// TwinCAT 3 PLC project Untitled1
// ProgramVersion: 3.1.4023.0
// CompilerDefines: VISU_USEWSTRING
// libraries:
//   CmpBitmapPool, * (System)
//   Tc2_Standard, * (Beckhoff Automation GmbH)
//   Tc2_System, * (Beckhoff Automation GmbH)
//   Tc3_Module, * (Beckhoff Automation GmbH)
//   VisuDialogs, * (System)
//   MachineManage,newest,Secote
// project tree:
//   DUTs/ E_Axis.TcDUT, E_Cylinder.TcDUT, E_Line.TcDUT, E_LineClose.TcDUT, E_LoadClose.TcDUT, E_LoadPriority.TcDUT, E_MachineType.TcDUT, E_Station.TcDUT, E_TakeMode.TcDUT, ST_Input.TcDUT, ST_Output.TcDUT, ST_Recipe.TcDUT, ST_Setting.TcDUT
//   DUTs/Station/Dismantling/ ST_StationDismantling.TcDUT, ST_StationDismantlingHandshake.TcDUT
//   DUTs/Station/ E_StationState.TcDUT, ST_StationHandshake.TcDUT, ST_StationParameter.TcDUT
//   DUTs/Station/Line0Buffer/ ST_StationLine0Buffer.TcDUT, ST_StationLine0BufferHandshake.TcDUT
//   DUTs/Station/Line0Load/ ST_StationLine0Load.TcDUT, ST_StationLine0LoadHandshake.TcDUT
//   DUTs/Station/LineLoad/ ST_StationLineLoad.TcDUT, ST_StationLineLoadHandshake.TcDUT
//   DUTs/Station/TakeLoad/ ST_StationTakeLoad.TcDUT, ST_StationTakeLoadHandshake.TcDUT
//   DUTs/Station/UnloadElevator/ ST_StationUnloadElevator.TcDUT, ST_StationUnloadElevatorHandshake.TcDUT
//   DUTs/Station/UnloadLine/ ST_StationUnloadLine.TcDUT, ST_StationUnloadLineHandshake.TcDUT
//   DUTs/Station/UnloadUc/ ST_StationUnloadUc.TcDUT, ST_StationUnloadUcHandshake.TcDUT
//   DUTs/Station/UnloadUc_311/ ST_StationUnloadUc_311.TcDUT, ST_StationUnloadUc_311Handshake.TcDUT
//   / GlobalTextList.TcGTLO, PlcTask.TcTTO, RecipeManager.TcRMO (not stored), VISU_TASK.TcTTO, 视图管理器.TcVMO (not stored)
//   GVLs/ GVL.TcGVL, GVL_Data.TcGVL, GVL_IO.TcGVL
//   POUs/Device/ FB_LineAxis.TcPOU
//   POUs/ MAIN.TcPOU, P_Alarm.TcPOU, P_Device.TcPOU, P_Station.TcPOU, P_System.TcPOU
//   POUs/Station/ FB_StationDismantling.TcPOU, FB_StationLine0Buffer.TcPOU, FB_StationLine0Load.TcPOU, FB_StationLineLoad.TcPOU, FB_StationTakeLoad.TcPOU, FB_StationUnloadElevator.TcPOU, FB_StationUnloadLine.TcPOU, FB_StationUnloadUc.TcPOU, FB_StationUnLoadUc_311.TcPOU
//   VISUs/Ctrl/ CtrlLine.TcVIS, CtrlOther.TcVIS, CtrlOutput.TcVIS, CtrlInput.TcVIS, FrameMain.TcVIS
//   VISUs/Image/ ImagePool.TcIPO (not stored)
//   VISUs/ PageData.TcVIS, PageHome.TcVIS, PageMessage.TcVIS, PageMonitor.TcVIS, PageSetting.TcVIS
//   VISUs/Text/ InputText.TcTLO, LineClose.TcTLO, LineLoadClose.TcTLO, LoadPriority.TcTLO, MachineType.TcTLO, ManualText.TcTLO, OutputText.TcTLO

CONFIGURATION Untitled1
    RESOURCE PLC ON TwinCAT3
        TASK PlcTask(INTERVAL := T#2ms, PRIORITY := 20);
        TASK VISU_TASK(INTERVAL := T#50000us, PRIORITY := 30);
        PROGRAM MAIN WITH PlcTask : MAIN;
        PROGRAM VisuElems_Visu_Prg WITH VISU_TASK : VisuElems.Visu_Prg;
    END_RESOURCE
END_CONFIGURATION

// ---- DUTs/E_Axis.TcDUT
{attribute 'qualified_only'}
{attribute 'strict'}
TYPE E_Axis :
(
	TakeY:=1,
	TakeZ,
	UC_Y
);
END_TYPE

// ---- DUTs/E_Cylinder.TcDUT
{attribute 'qualified_only'}
{attribute 'strict'}
TYPE E_Cylinder :
(
Line0Part:=1,//主流线分料气缸

Line0Prevent,//主流线阻挡气缸

Line1Elevator,//流水线1提升气缸

Line1Lift,//流水线1顶升气缸

Line1Prevent,//流水线1阻挡气缸

Line1Rotate,//流水线1旋转气缸

Line1Adjust1,//流水线1调宽气缸1

Line2Lift,//流水线2顶升气缸

Line2Prevent,//流水线2阻挡气缸

Line2Standard1,//流水线2校平气缸1

Line2Standard2,//流水线2校平气缸2

Line2OpenLateral1,//流水线2解锁侧推气缸1

Line2OpenRotate,//流水线2解锁旋转气缸

Line2OpenLateral2,//流水线2解锁侧推气缸2

Line3LoadLift,//流水线3上料位顶升

Line3LoadPrevent,//流水线3上料位阻挡

Line3LoadRotate,//流水线3上料位旋转

Line3OpenLift,//流水线3解锁位顶升

Line3OpenPrevent,//流水线3解锁位阻挡

Line3Standard1,//流水线3校平气缸1

Line3Standard2,//流水线3校平气缸2

Line3OpenLateral1,//流水线3解锁侧推气缸1

Line3OpenRotate,//流水线3解锁旋转气缸

Line3OpenLateral2,//流水线3解锁侧推气缸2

TakeLift1,//取料模组升降气缸1

TakeLift2,//取料模组升降气缸2

TakeClamp,//取料模组夹紧气缸

UcLift,//下UC模组升降气缸

UcClamp,//下UC模组夹紧气缸

UcSwing,//下UC模组摆动气缸

UcLift1,//下UC升降气缸1

UcClamp1,//下UC夹紧气缸1

UcRotate1,//下UC旋转气缸1

UcLift2,//下UC升降气缸2

UcClamp2,//下UC夹紧气缸2

UcRotate2,//下UC旋转气缸2

UcDrive,//下UC皮带推料气缸

FrockElevator1,//下工装提升气缸1

FrockRotateDown1,//下工装旋转压紧气缸1

FrockPush1,//下工装拨料气缸1

FrockElevator2,//下工装提升气缸2

FrockRotateDown2,//下工装旋转压紧气缸2

FrockPush2,//下工装拨料气缸2

FrockBelt//下工装皮带推料气缸
);
END_TYPE

// ---- DUTs/E_Line.TcDUT
{attribute 'qualified_only'}
{attribute 'strict'}
TYPE E_Line :
(
	UnloadElevator := 1,
	UnloadUC,
	Line1,
	Line2,
	Line3
	
);
END_TYPE

// ---- DUTs/E_LineClose.TcDUT
{attribute 'qualified_only'}
{attribute 'strict'}
TYPE E_LineClose :
(
	None := 0,
	Line2,
	Line3
);
END_TYPE

// ---- DUTs/E_LoadClose.TcDUT
{attribute 'qualified_only'}
{attribute 'strict'}
TYPE E_LoadClose :
(
	None:=0,// 不关闭
	Line0,
	Line1
);
END_TYPE

// ---- DUTs/E_LoadPriority.TcDUT
{attribute 'qualified_only'}
{attribute 'strict'}
TYPE E_LoadPriority :
(
	None := 0,// 无等级
	Line0,// 优先0
	Line1// 优先1
);
END_TYPE

// ---- DUTs/E_MachineType.TcDUT
{attribute 'qualified_only'}
{attribute 'strict'}
TYPE E_MachineType :
(
	None:=0,
	RH353,
	RH367,
	RH311,
	RH201,
	RH069,
	RH373,
	LH353,
	LH367,
	LH311,
	LH201,
	LH069,
	LH373
);
END_TYPE

// ---- DUTs/E_Station.TcDUT
{attribute 'qualified_only'}
{attribute 'strict'}
TYPE E_Station :
(
	Line0Load:=0,// 主流线上料工站
	Line0Buffer,// 主流线缓存工站
	TakeLoad,// 上料取料工站
	Line3Load,// 流线3上料工站
	Line1Load,// 流线2上料工站
	Line2Dismantling,// 流线2拆解工站
	Line3Dismantling,// 流线3拆解工站
	Line2UnloadElevator,// 线体2下工装
	Line3UnloadElevator,// 线体3下工装
	Line2UnloadUc,// 线体2 下UC
	Line3UnloadUc,// 线体2 下UC
	UnloadLineUc,// 下UC 线体
	UnloadLineElevator,// 下工装 线体
	UnloadUc_311,// 下UC模组
	Length
);
END_TYPE

// ---- DUTs/E_TakeMode.TcDUT
{attribute 'qualified_only'}
{attribute 'strict'}
TYPE E_TakeMode :
(
	None := 0,// 不动作
	Take0,// 取Line0料
	Take1,// 取Line1料
	Take3Load,// 取Line3上料站 产品
	Place1,// 放Line1料
	Place3Load// 放线体3上料站
);
END_TYPE

// ---- DUTs/Station/Dismantling/ST_StationDismantling.TcDUT
TYPE ST_StationDismantling :
STRUCT
	fbLift:				 	REFERENCE TO FB_Cylinder;// 顶升气缸
	fbPrevent:				REFERENCE TO FB_Cylinder;// 阻挡气缸
	fbStandard1:			REFERENCE TO FB_Cylinder;// 校平气缸1
	fbStandard2:			REFERENCE TO FB_Cylinder;// 校平气缸2
	fbLateral1:				REFERENCE TO FB_Cylinder;// 侧推气缸1
	fbLateral2:				REFERENCE TO FB_Cylinder;// 侧推气缸2
	fbRotate:				REFERENCE TO FB_Cylinder;// 旋转气缸
	bPalletCheck1:			BOOL;// 流入光电
	bPalletCheck2:			BOOL;// 到位光电
	bPalletCheck3:			BOOL;// 流出光电
	eState:					E_StationState;
	bClose:					BOOL;// 关闭线体
	bCloseUnloadElevator:	BOOL;// 关闭下工装
	stHandshake:			ST_StationDismantlingHandshake;
END_STRUCT
END_TYPE

// ---- DUTs/Station/Dismantling/ST_StationDismantlingHandshake.TcDUT
TYPE ST_StationDismantlingHandshake :
STRUCT
	bRequestLineLoad_D:			BOOL;// 拆解工站 请求上料 只写
	bResponseDismantling_D:		BOOL;// 收到 拆解工站 请求上料 只读
	
	bRequestUc:					BOOL;// 拆解站 向下UC站 请求放料 只写
	bResponseDismantling_Uc:	BOOL;// 收到 拆解站 向下UC站 请求放料 只读
	
	bRequestElevator:			BOOL;// 拆解站 向下工装 请求放料 只写
	bResponseDismantling_E:		BOOL;// 收到 拆解站 向下工装站 请求放料 只读
	
END_STRUCT
END_TYPE

// ---- DUTs/Station/E_StationState.TcDUT
{attribute 'qualified_only'}
{attribute 'strict'}
TYPE E_StationState :
(
	None:=0,
	Load,// 等待上料
	Busy,// 工作中
	Done// 工作完成
);
END_TYPE

// ---- DUTs/Station/Line0Buffer/ST_StationLine0Buffer.TcDUT
TYPE ST_StationLine0Buffer :
STRUCT
	bPlace:				BOOL;// 到位光电
	eState:				E_StationState;
	stHandshake:		ST_StationLine0BufferHandshake;
END_STRUCT
END_TYPE

// ---- DUTs/Station/Line0Buffer/ST_StationLine0BufferHandshake.TcDUT
TYPE ST_StationLine0BufferHandshake :
STRUCT
	bRequestLine0Load:			BOOL;// 请求线体0 上料站 放料 只写
	bResponseLine0Buffer:		BOOL;// 收到线体0 上料缓存站 放料请求 只读
	
	bRequestLine0Buffer_T:		BOOL;// 取料站 向线体0 请求 取料 只读
	bResponseTake_T:			BOOL;// 收到 取料站 取料请求 只写
END_STRUCT
END_TYPE

// ---- DUTs/Station/Line0Load/ST_StationLine0Load.TcDUT
TYPE ST_StationLine0Load :
STRUCT
	fbPart:			REFERENCE TO FB_Cylinder;// 分料气缸
	fbPrevent:		REFERENCE TO FB_Cylinder;// 阻挡气缸
	bPartCheck:		BOOL;// 分料光电
	bPreventCheck:	BOOL;// 阻挡光电
	stHandshake:	ST_StationLine0LoadHandshake;	
END_STRUCT
END_TYPE

// ---- DUTs/Station/Line0Load/ST_StationLine0LoadHandshake.TcDUT
TYPE ST_StationLine0LoadHandshake :
STRUCT
	bRequestLine0Load:			BOOL;// 请求线体0 上料站 放料 只读
	bResponseLine0Buffer:		BOOL;// 收到线体0 上料缓存站 放料请求 只写
END_STRUCT
END_TYPE

// ---- DUTs/Station/LineLoad/ST_StationLineLoad.TcDUT
TYPE ST_StationLineLoad :
STRUCT
	fbElevator:				REFERENCE TO FB_Cylinder;// 提升气缸
	fbLift:					REFERENCE TO FB_Cylinder;// 顶升气缸
	fbPrevent:				REFERENCE TO FB_Cylinder;// 阻挡气缸
	fbRotate:				REFERENCE TO FB_Cylinder;// 旋转气缸
	fbAdjust1:				REFERENCE TO FB_Cylinder;// 调宽气缸
	bPalletCheck1:			BOOL;// 流入光电
	bPalletCheck2:			BOOL;// 到位光电
	bPalletCheck3:			BOOL;// 流出光电
	eState:					E_StationState;
	bIsClosed:				BOOL;// 线体关闭
	bIsTaking:				BOOL;// 取料站 取料中
	bIsPlacing:				BOOL;// 取料站 放料中
	bManualLoad:			BOOL;// 手动上料 
	stHandshake:			ST_StationLineLoadHandshake;
END_STRUCT
END_TYPE

// ---- DUTs/Station/LineLoad/ST_StationLineLoadHandshake.TcDUT
TYPE ST_StationLineLoadHandshake :
STRUCT
	bRequestLineLoad_T:			BOOL;// 取料站 请求取料 只读
	bResponseTake_T:			BOOL;// 收到 取料站 请求取料 只写
	
	bRequestLineLoad_P:			BOOL;// 取料站 请求放料 只读
	bResponseTake_P:			BOOL;// 收到 取料站 请求放料 只写
	
	bRequestTake_P_M:			BOOL;// 上游设备 请求放料 只读
	bResponseMachine_P:			BOOL;// 收到 上游设备 请求放料 只写
	
	bRequestLineLoad_D:			BOOL;// 拆解工站 请求上料 只读
	bResponseDismantling_D:		BOOL;// 收到 拆解工站 请求上料 只写
END_STRUCT
END_TYPE

// ---- DUTs/Station/ST_StationHandshake.TcDUT
TYPE ST_StationHandshake :
STRUCT
	(*bLine0BufferRequestLine0Load:			BOOL;// Line0缓存站 请求上料站放料
	bLine0LoadResponseLine0Buffer:			BOOL;// line0上料站 收到缓存站请求
	

	arrRequestTaskLine:						ARRAY[0..2] OF	BOOL;// 请求取线体上料站 产品 0:Lin0 1:Line1 2:Lin3Load
	arrRequestPlaceLine:					ARRAY[1..2] OF	BOOL;// 请求往线体上料站 放料 1:Line1 2:Lin3Load
	
	arrResponseTaskLine:					ARRAY[0..2] OF	BOOL;// 线体上料站收到取料请求 0:Lin0 1:Line1 2:Lin3Load
	arrResponsePlaceLine:					ARRAY[1..2] OF 	BOOL;// 线体上料站收到放料请求 1:Line1 2:Lin3Load
	
	
	bLoadMachineReady:					    BOOL;// Line1对接设备准备就绪
	bLoadMachineReadyOk:					BOOL;// 收到Line1对接设备请求信号
	
	arrDismantlingRequest:					ARRAY[1..2] OF BOOL;// 拆解站请求放料 1:Line2 2:Lin3
	arrDismantlingResponse:					ARRAY[1..2] OF BOOL;// 上料站收到拆解站请求信号 1:Line1 2:Lin3
	
	arrDismantlingRequestUc:				ARRAY[1..2] OF BOOL;// 拆解站请求取Uc 1:Line2 2:Lin3
	arrDismantlingResponseUc:				ARRAY[1..2] OF BOOL;// 收到拆解站请求取Uc 1:Line2 2:Lin3
	
	arrUnloadUcRequest:						ARRAY[1..2] OF BOOL;// 下UC工站 请求放料
	arrUnloadUcResponse:					ARRAY[1..2] OF BOOL;// 下UC线体 收到放料请求
	
	arrUnloadElevatorRequest:				ARRAY[1..2] OF BOOL;// 下UC工站 请求放料
	arrUnloadElevatorResponse:				ARRAY[1..2] OF BOOL;// 下UC线体 收到放料请求*)
END_STRUCT
END_TYPE

// ---- DUTs/Station/ST_StationParameter.TcDUT
TYPE ST_StationParameter :
STRUCT
	stLine0Load:			ST_StationLine0Load;// 主流线上料工站
	stLine0Buffer:			ST_StationLine0Buffer;// 主流线缓存工站
	stTakeLoad:				ST_StationTakeLoad;// 上料取料工站
	stLine3Load:			ST_StationLineLoad;// 流线3上料工站
	stLine1Load:			ST_StationLineLoad;// 流线2上料工站
	stLine2Dismantling:		ST_StationDismantling;// 流线2拆解工站
	stLine3Dismantling:		ST_StationDismantling;// 流线3拆解工站
	stLine2UnloadElevator:	ST_StationUnloadElevator;// 线体2下工装
	stLine3UnloadElevator:	ST_StationUnloadElevator;// 线体3下工装
	stLine2UnloadUc:		ST_StationUnloadUc;// 线体2 下UC
	stLine3UnloadUc:		ST_StationUnloadUc;// 线体2 下UC
	stUnloadLineUc:			ST_StationUnloadLine;// 下UC 线体
	stUnloadLineElevator:	ST_StationUnloadLine;// 下工装 线体
	stUnloadUc_311:			ST_StationUnloadUc_311;// 下UC 模组
END_STRUCT
END_TYPE

// ---- DUTs/Station/TakeLoad/ST_StationTakeLoad.TcDUT
TYPE ST_StationTakeLoad :
STRUCT
	fbTakeLift1:		REFERENCE TO FB_Cylinder;// 升降气缸1
	fbTakeLift2:		REFERENCE TO FB_Cylinder;// 升降气缸2
	fbTakeClamp:		REFERENCE TO FB_Cylinder;// 加紧气缸
	fbTakeZ:			REFERENCE TO FB_Axis;// Z轴
	fbTakeY:			REFERENCE TO FB_Axis;// Y轴
	eState:				E_StationState;
	stHandshake:		ST_StationTakeLoadHandshake;
END_STRUCT
END_TYPE

// ---- DUTs/Station/TakeLoad/ST_StationTakeLoadHandshake.TcDUT
TYPE ST_StationTakeLoadHandshake :
STRUCT
	bRequestLine0Buffer_T0:		BOOL;// 取料站 向线体0 请求 取料 只写
	bResponseTake_T0:			BOOL;// 收到 取料站 取料请求 只读
	
	bRequestLineLoad_T1:	BOOL;// 取料站 请求取料 Line1 只写
	bResponseTake_T1:		BOOL;// 收到 取料站 请求取料 Line1 只读
	
	bRequestLineLoad_T3:	BOOL;// 取料站 请求取料 Line2 只写
	bResponseTake_T3:		BOOL;// 收到 取料站 请求取料 Line3 只读
	
	bRequestLineLoad_P3:	BOOL;// 取料站 请求放料 Lin3 只写
	bResponseTake_P3:		BOOL;// 收到 取料站 请求放料 Line3 只读
	
	bRequestLineLoad_P1:	BOOL;// 取料站 请求放料 Lin1 只写
	bResponseTake_P1:		BOOL;// 收到 取料站 请求放料 Line1 只读
END_STRUCT
END_TYPE

// ---- DUTs/Station/UnloadElevator/ST_StationUnloadElevator.TcDUT
TYPE ST_StationUnloadElevator :
STRUCT
	bFrockElevator1NoneCheck:			BOOL;//工装有无检测
	fbFrockElevator:					REFERENCE TO FB_Cylinder;// 提升气缸
	fbFrockRotateDown:					REFERENCE TO FB_Cylinder;// 旋转压紧气缸
	fbFrockPush:						REFERENCE TO FB_Cylinder;// 拨料气缸
	bManualUnload:						BOOL;// 手动下料
	stHandshake:						ST_StationUnloadElevatorHandshake;
END_STRUCT
END_TYPE

// ---- DUTs/Station/UnloadElevator/ST_StationUnloadElevatorHandshake.TcDUT
TYPE ST_StationUnloadElevatorHandshake :
STRUCT
	bRequestElevator:			BOOL;// 拆解站 向下工装 请求放料 只读
	bResponseDismantling_E:		BOOL;// 收到 拆解站 向下工装站 请求放料 只写
	
	bRequestUnline:				BOOL;// 下工装 向下线体 请求放料 只写 
	bResponseElevator:			BOOL;// 收到 下工装 向下线体 请求放料 只读
END_STRUCT
END_TYPE

// ---- DUTs/Station/UnloadLine/ST_StationUnloadLine.TcDUT
TYPE ST_StationUnloadLine :
STRUCT
	fbDrive:				REFERENCE TO FB_Cylinder;// 推料气缸
	fbLineAxis:             REFERENCE TO FB_LineAxis;// 线体
	bCheck1:				BOOL;//有无检测1
	bCheck2:				BOOL;//有无检测2
	bBeltDone:				BOOL;//到位检测
	bBeltNoneCheck:			BOOL;//斜坡有无检测 
	bManualUnload:			BOOL;// 手动下料
	stHandshake:			ST_StationUnloadLineHandshake;
END_STRUCT
END_TYPE

// ---- DUTs/Station/UnloadLine/ST_StationUnloadLineHandshake.TcDUT
TYPE ST_StationUnloadLineHandshake :
STRUCT
	bRequestUnloadLine2:			BOOL;// 向下线体 请求放料 只读
	bResponseUnladLine2:			BOOL;//  收到 向下线体 请求放料 只写
	
	bRequestUnloadLine3:			BOOL;// 向下线体 请求放料 只读
	bResponseUnladLine3:			BOOL;//  收到 向下线体 请求放料 只写
END_STRUCT
END_TYPE

// ---- DUTs/Station/UnloadUc/ST_StationUnloadUc.TcDUT
TYPE ST_StationUnloadUc :
STRUCT
	fbLift:				REFERENCE TO FB_Cylinder;// 升降气缸
	fbClamp:			REFERENCE TO FB_Cylinder;// 夹紧气缸
	fbRotate:			REFERENCE TO FB_Cylinder;// 旋转气缸
	stHandshake:		ST_StationUnloadUcHandshake;
END_STRUCT
END_TYPE

// ---- DUTs/Station/UnloadUc/ST_StationUnloadUcHandshake.TcDUT
TYPE ST_StationUnloadUcHandshake :
STRUCT
	bRequestUc:					BOOL;// 拆解站 向下UC站 请求放料 只读
	bResponseDismantling_Uc:	BOOL;// 收到 拆解站 向下UC站 请求放料 只写
	
	bRequestUnloadLine:			BOOL;// 向下线体 请求放料 只写
	bResponseUnladLine:			BOOL;//  收到 向下线体 请求放料 只读
END_STRUCT
END_TYPE

// ---- DUTs/Station/UnloadUc_311/ST_StationUnloadUc_311.TcDUT
TYPE ST_StationUnloadUc_311 :
STRUCT
	bUcCheck1:					BOOL;// 下UC模组UC有无检测
	fbLift:						REFERENCE TO FB_Cylinder;// 下UC模组升降气缸
	fbClamp:					REFERENCE TO FB_Cylinder;// 下UC模组夹紧气缸
	fbSwing:					REFERENCE TO FB_Cylinder;// 下UC模组摆动气缸
	fbAxisY:					REFERENCE TO FB_Axis;// 取料Y轴
	stHandshake:				ST_StationUnloadUc_311Handshake;
END_STRUCT
END_TYPE

// ---- DUTs/Station/UnloadUc_311/ST_StationUnloadUc_311Handshake.TcDUT
TYPE ST_StationUnloadUc_311Handshake :
STRUCT
	bRequestUc_L2:					BOOL;// 拆解站 向下UC站 请求放料 只读
	bResponseDismantling_Uc_L2:		BOOL;// 收到 拆解站 向下UC站 请求放料 只写
	
	bRequestUc_L3:					BOOL;// 拆解站 向下UC站 请求放料 只读
	bResponseDismantling_Uc_L3:		BOOL;// 收到 拆解站 向下UC站 请求放料 只写
END_STRUCT
END_TYPE

// ---- DUTs/ST_Input.TcDUT
TYPE ST_Input :
STRUCT
bStart:BOOL;//启动 IN00
bStop:bool;//停止 IN01
bResetAlarm:bool;//报警复位 IN02
bEStop:bool;//急停 IN03
bDoor:bool;//安全门开关 IN04
bNone1:bool;//预留 IN05
bNone2:bool;//预留 IN06
bLine0Part_Cyl_H:bool;//主流线分料气缸原位 IN07
bLine0Part_Cyl_W:bool;//主流线分料气缸工作位 IN08
bLine0Prevent_Cyl_H:bool;//主流线阻挡气缸原位 IN09
bLine0Prevent_Cyl_W:bool;//主流线阻挡气缸工作位 IN0A
bLine1Elevator_Cyl_H:bool;//流水线1提升气缸原位 IN0B
bLine1Elevator_Cyl_W:bool;//流水线1提升气缸工作位 IN0C
bLine1Lift_Cyl_H:bool;//流水线1顶升气缸原位 IN0D
bLine1Lift_Cyl_W:bool;//流水线1顶升气缸工作位 IN0E
bLine1Prevent_Cyl_H:bool;//流水线1阻挡气缸原位 IN0F
bLine1Prevent_Cyl_W:bool;//流水线1阻挡气缸工作位 IN10
bLine1Rotate_Cyl_H:bool;//流水线1旋转气缸原位 IN11
bLine1Rotate_Cyl_W:bool;//流水线1旋转气缸工作位 IN12
bLine1Adjust1_Cyl_H:bool;//流水线1调宽气缸原位1 IN13
bLine1Adjust1_Cyl_W:bool;//流水线1调宽气缸工作位1 IN14
bLine1Adjust2_Cyl_H:bool;//流水线1调宽气缸原位2 IN15
bLine1Adjust2_Cyl_W:bool;//流水线1调宽气缸工作位2 IN16
bLine2Lift_Cyl_H:bool;//流水线2顶升气缸原位 IN17
bLine2Lift_Cyl_W:bool;//流水线2顶升气缸工作位 IN18
bLine2Prevent_Cyl_H:bool;//流水线2阻挡气缸原位 IN19
bLine2Prevent_Cyl_W:bool;//流水线2阻挡气缸工作位 IN1A
bLine2Standard1_Cyl_H:bool;//流水线2校平气缸1原位 IN1B
bLine2Standard1_Cyl_W:bool;//流水线2校平气缸1工作位 IN1C
bLine2Standard2_Cyl_H:bool;//流水线2校平气缸2原位 IN1D
bLine2Standard2_Cyl_W:bool;//流水线2校平气缸2工作位 IN1E
bLine2OpenLateral1_Cyl_H:bool;//流水线2解锁侧推气缸1原位 IN1F
bLine2OpenLateral1_Cyl_W:bool;//流水线2解锁侧推气缸1工作位 IN20
bLine2OpenRotate_Cyl_H:bool;//流水线2解锁旋转气缸原位 IN21
bLine2OpenRotate_Cyl_W:bool;//流水线2解锁旋转气缸工作位 IN22
bLine2OpenLateral2_Cyl_H:bool;//流水线2解锁侧推气缸2原位 IN23
bLine2OpenLateral2_Cyl_W:bool;//流水线2解锁侧推气缸2工作位 IN24
None:bool;//空 IN25
None1:bool;//空 IN26
bLine3LoadLift_Cyl_H:bool;//流水线3上料位顶升原位 IN27
bLine3LoadLift_Cyl_W:bool;//流水线3上料位顶升工作位 IN28
bLine3LoadPrevent_Cyl_H:bool;//流水线3上料位阻挡原位 IN29
bLine3LoadPrevent_Cyl_W:bool;//流水线3上料位阻挡工作位 IN2A
bLine3LoadRotate_Cyl_H:bool;//流水线3上料位旋转原位 IN2B
bLine3LoadRotate_Cyl_W:bool;//流水线3上料位旋转工作位 IN2C
bLine3OpenLift_Cyl_H:bool;//流水线3解锁位顶升原位 IN2D
bLine3OpenLift_Cyl_W:bool;//流水线3解锁位顶升工作位 IN2E
bLine3OpenPrevent_Cyl_H:bool;//流水线3解锁位阻挡原位 IN2F
bLine3OpenPrevent_Cyl_W:bool;//流水线3解锁位阻挡工作位 IN30
bLine3Standard1_Cyl_H:bool;//流水线3校平气缸1原位 IN31
bLine3Standard1_Cyl_W:bool;//流水线3校平气缸1工作位 IN32
bLine3Standard2_Cyl_H:bool;//流水线3校平气缸2原位 IN33
bLine3Standard2_Cyl_W:bool;//流水线3校平气缸2工作位 IN34
bLine3OpenLateral1_Cyl_H:bool;//流水线3解锁侧推气缸1原位 IN35
bLine3OpenLateral1_Cyl_W:bool;//流水线3解锁侧推气缸1工作位 IN36
bLine3OpenRotate_Cyl_H:bool;//流水线3解锁旋转气缸原位 IN37
bLine3OpenRotate_Cyl_W:bool;//流水线3解锁旋转气缸工作位 IN38
bLine3OpenLateral2_Cyl_H:bool;//流水线3解锁侧推气缸2原位 IN39
bLine3OpenLateral2_Cyl_W:bool;//流水线3解锁侧推气缸2工作位 IN3A
None3:bool;//空 IN3B
None4:bool;//空 IN3C
bTakeLift1_Cyl_H:bool;//取料模组升降气缸1原位 IN3D
bTakeLift1_Cyl_W:bool;//取料模组升降气缸1工作位 IN3E
bTakeLift2_Cyl_H:bool;//取料模组升降气缸2原位 IN3F
bTakeLift2_Cyl_W:bool;//取料模组升降气缸2工作位 IN40
bTakeClamp_Cyl_H:bool;//取料模组夹紧气缸原位 IN41
bTakeClamp_Cyl_W:bool;//取料模组夹紧气缸工作位 IN42
bUcLift_Cyl_H:bool;//下UC模组升降气缸原位 IN43
bUcLift_Cyl_W:bool;//下UC模组升降气缸工作位 IN44
bUcClamp_Cyl_H:bool;//下UC模组夹紧气缸原位 IN45
bUcClamp_Cyl_W:bool;//下UC模组夹紧气缸工作位 IN46
bUcSwing_Cyl_H:bool;//下UC模组摆动气缸原位 IN47
bUcSwing_Cyl_W:bool;//下UC模组摆动气缸工作位 IN48
bUcLift1_Cyl_H:bool;//下UC升降气缸1原位 IN49
bUcLift1_Cyl_W:bool;//下UC升降气缸1工作位 IN4A
bUcClamp1_Cyl_H:bool;//下UC夹紧气缸1原位 IN4B
bUcClamp1_Cyl_W:bool;//下UC夹紧气缸1工作位 IN4C
bUcRotate1_Cyl_H:bool;//下UC旋转气缸1原位 IN4D
bUcRotate1_Cyl_W:bool;//下UC旋转气缸1工作位 IN4E
bUcLift2_Cyl_H:bool;//下UC升降气缸2原位 IN4F
bUcLift2_Cyl_W:bool;//下UC升降气缸2工作位 IN50
bUcClamp2_Cyl_H:bool;//下UC夹紧气缸2原位 IN51
bUcClamp2_Cyl_W:bool;//下UC夹紧气缸2工作位 IN52
bUcRotate2_Cyl_H:bool;//下UC旋转气缸2原位 IN53
bUcRotate2_Cyl_W:bool;//下UC旋转气缸2工作位 IN54
bUcDrive_Cyl_H:bool;//下UC皮带推料气缸原位 IN55
bUcDrive_Cyl_W:bool;//下UC皮带推料气缸工作位 IN56
bFrockElevator1_Cyl_H:bool;//下工装提升气缸1原位 IN57
bFrockElevator1_Cyl_W:bool;//下工装提升气缸1工作位 IN58
bFrockRotateDown1_Cyl_H:bool;//下工装旋转压紧气缸1原位 IN59
bFrockRotateDown1_Cyl_W:bool;//下工装旋转压紧气缸1工作位 IN5A
bFrockPush1_Cyl_H:bool;//下工装拨料气缸1原位 IN5B
bFrockPush1_Cyl_W:bool;//下工装拨料气缸1工作位 IN5C
bFrockElevator2_Cyl_H:bool;//下工装提升气缸2原位 IN5D
bFrockElevator2_Cyl_W:bool;//下工装提升气缸2工作位 IN5E
bFrockRotateDown2_Cyl_H:bool;//下工装旋转压紧气缸2原位 IN5F
bFrockRotateDown2_Cyl_W:bool;//下工装旋转压紧气缸2工作位 IN60
bFrockPush2_Cyl_H:bool;//下工装拨料气缸2原位 IN61
bFrockPush2_Cyl_W:bool;//下工装拨料气缸2工作位 IN62
bFrockBelt_Cyl_H:bool;//下工装皮带推料气缸原位 IN63
bFrockBelt_Cyl_W:bool;//下工装皮带推料气缸工作位 IN64
bNone3:bool;//预留 IN65
bLine0Part:bool;//主流线分料光电 IN66
bLine0Prevent:bool;//主流线阻挡光电 IN67
bLine0Place:bool;//主流线到位光电 IN68
bLine1PalletCheck1:bool;//流水线1流入光电 IN69
bLine1PalletCheck2:bool;//流水线1到位光电 IN6A
bLine1PalletCheck3:bool;//流水线1流出光电 IN6B
bLine2PalletCheck1:bool;//流水线2流入光电 IN6C
bLine2PalletCheck2:bool;//流水线2到位光电 IN6D
bLine2PalletCheck3:bool;//流水线2流出光电 IN6E
bLine3PalletCheck1:bool;//流水线3上料位流入光电 IN6F
bLine3PalletCheck2:bool;//流水线3上料位到位光电 IN70
bLine3PalletCheck3:bool;//流水线3上料位流出光电 IN71
bLine3OpenCheck1:bool;//流水线3解锁位流入光电 IN72
bLine3OpenCheck2:bool;//流水线3解锁位到位光电 IN73
bLine3OpenCheck3:bool;//流水线3解锁位流出光电 IN74
bUcCheck1:bool;//下UC模组UC有无检测1 IN75
bUcCheck2:bool;//下UC皮带UC有无检测2 IN76
bUcCheck3:bool;//下UC皮带UC有无检测3 IN77
bUcBeltDone:bool;//下UC皮带到位检测 IN78
bUcBeltNoneCheck:bool;//下UC皮带斜坡有无检测 IN79
bFrockElevator1NoneCheck:bool;//下工装提升1工装有无检测 IN7A
bFrockElevator2NoneCheck:bool;//下工装提升2工装有无检测 IN7B
bFrockBeltNoneCheck1:bool;//下工装皮带工装有无检测1 IN7C
bFrockBeltNoneCheck2:bool;//下工装皮带工装有无检测2 IN7D
bFrockBeltDone:bool;//下工装皮带到位检测 IN7E
bFrockBeltNoneCheck3:bool;//下工装皮带斜坡有无检测 IN7F
END_STRUCT
END_TYPE

// ---- DUTs/ST_Output.TcDUT
TYPE ST_Output :
STRUCT
bBeacon_Red:BOOL;//三色灯红 OUT00
bBeacon_Yellow:bool;//三色灯黄 OUT01
bBeacon_Green:bool;//三色灯绿 OUT02
bBeacon_Buzzer:bool;//蜂鸣器 OUT03
bRuning:bool;//运行指示灯 OUT04
bStop:bool;//停止指示灯 OUT05
bLED:bool;//照明灯 OUT06
bLine0Part_Cyl_H:bool;//主流线分料气缸缩回 OUT07
bLine0Part_Cyl_W:bool;//主流线分料气缸伸出 OUT08
bLine0Prevent_Cyl_H:bool;//主流线阻挡气缸缩回 OUT09
bLine0Prevent_Cyl_W:bool;//主流线阻挡气缸伸出 OUT0A
bLine1Elevator_Cyl_H:bool;//流水线1提升气缸缩回 OUT0B
bLine1Elevator_Cyl_W:bool;//流水线1提升气缸伸出 OUT0C
bLine1Lift_Cyl_H:bool;//流水线1顶升气缸缩回 OUT0D
bLine1Lift_Cyl_W:bool;//流水线1顶升气缸伸出 OUT0E
bLine1Prevent_Cyl_H:bool;//流水线1阻挡气缸缩回 OUT0F
bLine1Prevent_Cyl_W:bool;//流水线1阻挡气缸伸出 OUT10
bLine1Rotate_Cyl_H:bool;//流水线1旋转气缸缩回 OUT11
bLine1Rotate_Cyl_W:bool;//流水线1旋转气缸伸出 OUT12
bLine1Adjust1_Cyl_H:bool;//流水线1调宽气缸缩回 OUT13
bLine1Adjust1_Cyl_W:bool;//流水线1调宽气缸伸出 OUT14
None1:bool;//预留 OUT15
None2:bool;//预留 OUT16
bLine2Lift_Cyl_H:bool;//流水线2顶升气缸缩回 OUT17
bLine2Lift_Cyl_W:bool;//流水线2顶升气缸伸出 OUT18
bLine2Prevent_Cyl_H:bool;//流水线2阻挡气缸缩回 OUT19
bLine2Prevent_Cyl_W:bool;//流水线2阻挡气缸伸出 OUT1A
bLine2Standard1_Cyl_H:bool;//流水线2校平气缸1缩回 OUT1B
bLine2Standard1_Cyl_W:bool;//流水线2校平气缸1伸出 OUT1C
bLine2Standard2_Cyl_H:bool;//流水线2校平气缸2缩回 OUT1D
bLine2Standard2_Cyl_W:bool;//流水线2校平气缸2伸出 OUT1E
bLine2OpenLateral1_Cyl_H:bool;//流水线2解锁侧推气缸1缩回 OUT1F
bLine2OpenLateral1_Cyl_W:bool;//流水线2解锁侧推气缸1伸出 OUT20
bLine2OpenRotate_Cyl_H:bool;//流水线2解锁旋转气缸缩回 OUT21
bLine2OpenRotate_Cyl_W:bool;//流水线2解锁旋转气缸伸出 OUT22
bLine2OpenLateral2_Cyl_H:bool;//流水线2解锁侧推气缸2缩回 OUT23
bLine2OpenLateral2_Cyl_W:bool;//流水线2解锁侧推气缸2伸出 OUT24
None202:bool;//预留 OUT25
None203:bool;//预留 OUT26
bLine3LoadLift_Cyl_H:bool;//流水线3上料位顶升缩回 OUT27
bLine3LoadLift_Cyl_W:bool;//流水线3上料位顶升伸出 OUT28
bLine3LoadPrevent_Cyl_H:bool;//流水线3上料位阻挡缩回 OUT29
bLine3LoadPrevent_Cyl_W:bool;//流水线3上料位阻挡伸出 OUT2A
bLine3LoadRotate_Cyl_H:bool;//流水线3上料位旋转缩回 OUT2B
bLine3LoadRotate_Cyl_W:bool;//流水线3上料位旋转伸出 OUT2C
bLine3OpenLift_Cyl_H:bool;//流水线3解锁位顶升缩回 OUT2D
bLine3OpenLift_Cyl_W:bool;//流水线3解锁位顶升伸出 OUT2E
bLine3OpenPrevent_Cyl_H:bool;//流水线3解锁位阻挡缩回 OUT2F
bLine3OpenPrevent_Cyl_W:bool;//流水线3解锁位阻挡伸出 OUT30
bLine3Standard1_Cyl_H:bool;//流水线3校平气缸1缩回 OUT31
bLine3Standard1_Cyl_W:bool;//流水线3校平气缸1伸出 OUT32
bLine3Standard2_Cyl_H:bool;//流水线3校平气缸2缩回 OUT33
bLine3Standard2_Cyl_W:bool;//流水线3校平气缸2伸出 OUT34
bLine3OpenLateral1_Cyl_H:bool;//流水线3解锁侧推气缸1缩回 OUT35
bLine3OpenLateral1_Cyl_W:bool;//流水线3解锁侧推气缸1伸出 OUT36
bLine3OpenRotate_Cyl_H:bool;//流水线3解锁旋转气缸缩回 OUT37
bLine3OpenRotate_Cyl_W:bool;//流水线3解锁旋转气缸伸出 OUT38
bLine3OpenLateral2_Cyl_H:bool;//流水线3解锁侧推气缸2缩回 OUT39
bLine3OpenLateral2_Cyl_W:bool;//流水线3解锁侧推气缸2伸出 OUT3A
None200:bool;//预留 OUT3B
None201:bool;//预留 OUT3C
bTakeLift1_Cyl_H:bool;//取料模组升降气缸1缩回 OUT3D
bTakeLift1_Cyl_W:bool;//取料模组升降气缸1伸出 OUT3E
bTakeLift2_Cyl_H:bool;//取料模组升降气缸2缩回 OUT3F
bTakeLift2_Cyl_W:bool;//取料模组升降气缸2伸出 OUT40
bTakeClamp_Cyl_H:bool;//取料模组夹紧气缸缩回 OUT41
bTakeClamp_Cyl_W:bool;//取料模组夹紧气缸伸出 OUT42
bUcLift_Cyl_H:bool;//下UC模组升降气缸缩回 OUT43
bUcLift_Cyl_W:bool;//下UC模组升降气缸伸出 OUT44
bUcClamp_Cyl_H:bool;//下UC模组夹紧气缸缩回 OUT45
bUcClamp_Cyl_W:bool;//下UC模组夹紧气缸伸出 OUT46
bUcSwing_Cyl_H:bool;//下UC模组摆动气缸缩回 OUT47
bUcSwing_Cyl_W:bool;//下UC模组摆动气缸伸出 OUT48
bUcLift1_Cyl_H:bool;//下UC升降气缸1缩回 OUT49
bUcLift1_Cyl_W:bool;//下UC升降气缸1伸出 OUT4A
bUcClamp1_Cyl_H:bool;//下UC夹紧气缸1缩回 OUT4B
bUcClamp1_Cyl_W:bool;//下UC夹紧气缸1伸出 OUT4C
bUcRotate1_Cyl_H:bool;//下UC旋转气缸1缩回 OUT4D
bUcRotate1_Cyl_W:bool;//下UC旋转气缸1伸出 OUT4E
bUcLift2_Cyl_H:bool;//下UC升降气缸2缩回 OUT4F
bUcLift2_Cyl_W:bool;//下UC升降气缸2伸出 OUT50
bUcClamp2_Cyl_H:bool;//下UC夹紧气缸2缩回 OUT51
bUcClamp2_Cyl_W:bool;//下UC夹紧气缸2伸出 OUT52
bUcRotate2_Cyl_H:bool;//下UC旋转气缸2缩回 OUT53
bUcRotate2_Cyl_W:bool;//下UC旋转气缸2伸出 OUT54
bUcDrive_Cyl_H:bool;//下UC皮带推料气缸缩回 OUT55
bUcDrive_Cyl_W:bool;//下UC皮带推料气缸伸出 OUT56
bFrockElevator1_Cyl_H:bool;//下工装提升气缸1缩回 OUT57
bFrockElevator1_Cyl_W:bool;//下工装提升气缸1伸出 OUT58
bFrockRotateDown1_Cyl_H:bool;//下工装旋转压紧气缸1缩回 OUT59
bFrockRotateDown1_Cyl_W:bool;//下工装旋转压紧气缸1伸出 OUT5A
bFrockPush1_Cyl_H:bool;//下工装拨料气缸1缩回 OUT5B
bFrockPush1_Cyl_W:bool;//下工装拨料气缸1伸出 OUT5C
bFrockElevator2_Cyl_H:bool;//下工装提升气缸2缩回 OUT5D
bFrockElevator2_Cyl_W:bool;//下工装提升气缸2伸出 OUT5E
bFrockRotateDown2_Cyl_H:bool;//下工装旋转压紧气缸2缩回 OUT5F
bFrockRotateDown2_Cyl_W:bool;//下工装旋转压紧气缸2伸出 OUT60
bFrockPush2_Cyl_H:bool;//下工装拨料气缸2缩回 OUT61
bFrockPush2_Cyl_W:bool;//下工装拨料气缸2伸出 OUT62
bFrockBelt_Cyl_H:bool;//下工装皮带推料气缸缩回 OUT63
bFrockBelt_Cyl_W:bool;//下工装皮带推料气缸伸出 OUT64
None3:bool;//预留 OUT65
bLine1Axis:bool;//流水线1皮带运行 OUT66
bLine2Axis:bool;//流水线2皮带运行 OUT67
bLine3Axis:bool;//流水线3皮带运行 OUT68
bUnloadUCLine:bool;//下UC皮带运行 OUT69
bUnloadElevatorLine:bool;//下工装皮带运行 OUT6A
None9:bool;//预留 OUT6B
None10:bool;//预留 OUT6C
None11:bool;//预留 OUT6D
None12:bool;//预留 OUT6E
None13:BOOL;//预留 OUT6F
END_STRUCT
END_TYPE

// ---- DUTs/ST_Recipe.TcDUT
TYPE ST_Recipe :
STRUCT
	eMachineType:				E_MachineType;// 设备类型
	eLoadPriority:				E_LoadPriority;// 上料优先级
	eLoadClose:					E_LoadClose;// 上料屏蔽
	eLineClose:					E_LineClose;// 屏蔽线体工位
	
	arrInputTon:				ARRAY[0..7,0..15] OF UINT;
	arrOutputTon:				ARRAY[0..6,0..15] OF UINT;
END_STRUCT
END_TYPE

// ---- DUTs/ST_Setting.TcDUT
TYPE ST_Setting :
STRUCT
	bDryRun:					BOOL;
	eTakeMode:					E_TakeMode;// 取料状态
	eTakeModeBuffer:			E_TakeMode;// 缓存取料状态
	tHomeLine:					TIME:=T#5S;// 初始化线体正转延迟
END_STRUCT
END_TYPE

// ---- GVLs/GVL.TcGVL
{attribute 'qualified_only'}
VAR_GLOBAL
	I:					ST_Input;// 输入信号
	Q:					ST_Output;// 输出信号
	stSetting:			ST_Setting;// 参数设置

	stShield_I:			ARRAY[0..7,0..15] OF  BOOL;;// 输入屏蔽
	stShield_Q:			ARRAY[0..6,0..15] OF  BOOL;//输出屏蔽

	arrFbLine:			ARRAY[0..10] OF FB_LineAxis;// 流线控制
END_VAR

// ---- GVLs/GVL_Data.TcGVL
{attribute 'qualified_only'}
VAR_GLOBAL PERSISTENT
	stRecipe:					ST_Recipe;// 配方
END_VAR

// ---- GVLs/GVL_IO.TcGVL
{attribute 'qualified_only'}
VAR_GLOBAL
	I AT %I*:				ARRAY[0..7,0..15] OF  BOOL;
	Q AT %Q*:				ARRAY[0..6,0..15] OF  BOOL;
	
	arrGetTorque AT %I*:	ARRAY[0..20] OF INT;
	arrSetTorque AT %Q*:	ARRAY[0..20] OF UINT;
	arrAxisInput AT %I*:	ARRAY[0..20] OF UDINT;
	
END_VAR

// ---- POUs/MAIN.TcPOU
PROGRAM MAIN
VAR
END_VAR

GVL_Data.stRecipe.eMachineType:=E_MachineType.RH069;
P_System();//系统程序
P_Alarm();// 报警程序
P_Device();// 外围装置
P_Station();// 工站流程

END_PROGRAM

// ---- POUs/P_System.TcPOU
PROGRAM P_System
VAR
	_arrFbButton:			ARRAY[0..10] OF FB_Button;
	
	_tonInit:				TON;
END_VAR

A_System();
A_Machine();

ACTION A_Machine:

END_ACTION

ACTION A_System:
G_stSystem.stInput.bEStop:=NOT GVL.I.bEStop;
G_stSystem.stInput.bInit:=GVL.I.bStart AND GVL.I.bStop;

//GVL.Q.bBeacon_Buzzer:=G_stSystem.stOutput.bBuzzer;
GVL.Q.bRuning:=GVL.Q.bBeacon_Green:=G_stSystem.stOutput.bLightGreen;
GVL.Q.bStop:=GVL.Q.bBeacon_Red:=G_stSystem.stOutput.bLightRed;
GVL.Q.bBeacon_Yellow:=G_stSystem.stOutput.bLightYellow;




_tonInit(IN:=GVL.I.bResetAlarm , PT:=T#5S , Q=> G_stSystem.stInput.bInit , ET=> );
_arrFbButton[0](In:=G_stSystem.stInput.bStart  , CLK:=GVL.I.bStart );
_arrFbButton[1](In:=G_stSystem.stInput.bStop  , CLK:=GVL.I.bStop );
_arrFbButton[2](In:=G_stSystem.stInput.bResetAlarm  , CLK:=GVL.I.bResetAlarm );


G_stSystem.stLogConfig.bExecute:=TRUE;
G_stSystem.stLogConfig.sFilePath:='D:\PLC\Log\System';

P_Machine(StationCount:=E_Station.Length);
END_ACTION

END_PROGRAM

// ---- POUs/P_Alarm.TcPOU
PROGRAM P_Alarm
VAR
	_arrFbErrorTag1:				ARRAY[0..20] OF  FB_ErrorTag;
	_arrFbErrorTag2:				ARRAY[0..20] OF  FB_ErrorTag;
	_arrFbErrorTag3:				ARRAY[0..20] OF  FB_ErrorTag;
	_arrFbErrorTag4:				ARRAY[0..20] OF  FB_ErrorTag;
	_arrFbErrorTag5:				ARRAY[0..20] OF  FB_ErrorTag;
	
	_i:								INT;
	
	_bFirstRun:						BOOL:=true;
END_VAR

G_stError.bSaveLog:=TRUE;
G_stError.sFileLogPath:='D:\PLC\Log\Error';

IF _bFirstRun THEN
	A_Info();
	_bFirstRun:=FALSE;
END_IF

A_Alarm1();
A_Alarm2();
A_Alarm3();
A_Alarm4();
A_Alarm5();

ACTION A_Alarm1:
_i:=0;
_arrFbErrorTag1[_i].Enable:=GVL_Data.stRecipe.eMachineType=E_MachineType.None;

_i:=1;
_arrFbErrorTag1[_i].Enable:=FALSE;//NOT GVL.I.bDoor;

_i:=2;
_arrFbErrorTag1[_i].Enable:=NOT GVL.I.bEStop;


FOR _i:=0 TO 20 BY 1 DO
_arrFbErrorTag1[_i](
	System:=G_stSystem , 
	Error:=G_stError , 
	ID:=TO_BYTE(_i+50) , 
	Category:=E_ErrorCategory.Safety , 
	InfoIndex:= , 
	Enable:= , 
	Message:= , 
	Level:=1 , 
	Position:="P_Alarm:A_Alarm1" , 
	ErrorTime:= , 
	Language:= , 
	Erroring=> , 
	ErrorCode=> );
END_FOR
END_ACTION

ACTION A_Alarm2:








FOR _i:=0 TO 20 BY 1 DO
_arrFbErrorTag2[_i](
	System:=G_stSystem , 
	Error:=G_stError , 
	ID:=TO_BYTE(52) , 
	Category:=E_ErrorCategory.Other , 
	InfoIndex:=TO_BYTE(_i) , 
	Enable:= , 
	Message:= , 
	Level:=2 , 
	Position:="P_Alarm:A_Alarm2" , 
	ErrorTime:= , 
	Language:= , 
	Erroring=> , 
	ErrorCode=> );
END_FOR
END_ACTION

ACTION A_Alarm3:
_i:=0;
_arrFbErrorTag3[_i].Enable:=G_stSystem.stMode.bAuto AND NOT G_stSystem.stMode.bHomeDone AND G_arrCylinder[E_Cylinder.TakeClamp].stOutput.bWork;



FOR _i:=0 TO 20 BY 1 DO
_arrFbErrorTag3[_i](
	System:=G_stSystem , 
	Error:=G_stError , 
	ID:=TO_BYTE(53) , 
	Category:=E_ErrorCategory.Other , 
	InfoIndex:=TO_BYTE(_i) , 
	Enable:= , 
	Message:= , 
	Level:=3 , 
	Position:="P_Alarm:A_Alarm3" , 
	ErrorTime:= , 
	Language:= , 
	Erroring=> , 
	ErrorCode=> );
END_FOR
END_ACTION

ACTION A_Alarm4:








FOR _i:=0 TO 20 BY 1 DO
_arrFbErrorTag4[_i](
	System:=G_stSystem , 
	Error:=G_stError , 
	ID:=TO_BYTE(54) , 
	Category:=E_ErrorCategory.Other , 
	InfoIndex:=TO_BYTE(_i) , 
	Enable:= , 
	Message:= , 
	Level:=4 , 
	Position:="P_Alarm:A_Alarm4" , 
	ErrorTime:= , 
	Language:= , 
	Erroring=> , 
	ErrorCode=> );
END_FOR
END_ACTION

ACTION A_Alarm5:









FOR _i:=0 TO 20 BY 1 DO
_arrFbErrorTag5[_i](
	System:=G_stSystem , 
	Error:=G_stError , 
	ID:=TO_BYTE(55) , 
	Category:=E_ErrorCategory.Other , 
	InfoIndex:=TO_BYTE(_i) , 
	Enable:= , 
	Message:= , 
	Level:=5 , 
	Position:="P_Alarm:A_Alarm5" , 
	ErrorTime:= , 
	Language:= , 
	Erroring=> , 
	ErrorCode=> );
END_FOR
END_ACTION

ACTION A_Info:
_arrFbErrorTag1[0].Language[E_Language.Chinese]:="设备类型为空 请选择设备类型";
_arrFbErrorTag1[0].Language[E_Language.English]:="Device type is empty please select device type";
_arrFbErrorTag1[0].Language[E_Language.Vietnamese]:="Thiết bị kiểu rỗng hãy chọn thiết bị kiểu";

_arrFbErrorTag1[1].Language[E_Language.Chinese]:="安全门未关闭";
_arrFbErrorTag1[1].Language[E_Language.English]:="The security door is open";
_arrFbErrorTag1[1].Language[E_Language.Vietnamese]:="Cửa an toàn chưa đóng";

_arrFbErrorTag1[2].Language[E_Language.Chinese]:="急停被按下";
_arrFbErrorTag1[2].Language[E_Language.English]:="Emergency stop is pressed";
_arrFbErrorTag1[2].Language[E_Language.Vietnamese]:="Dừng khẩn cấp bị nhấn";

_arrFbErrorTag3[0].Language[E_Language.Chinese]:="请确认取料夹爪是否有料 松开夹爪";
END_ACTION

END_PROGRAM

// ---- POUs/P_Device.TcPOU
PROGRAM P_Device
VAR
	_i:					INT;
	_t:					INT;
	
	_arrCylTon_H:		ARRAY[0..50] OF TON;
	_arrCylTon_W:		ARRAY[0..50] OF TON;
	_bFirstRun: 		BOOL:=TRUE;
	
	_arrInput :			ARRAY[0..7,0..15] OF  BOOL;
	_arrOutput:			ARRAY[0..6,0..15] OF  BOOL;
	
	_arrTonInput :		ARRAY[0..7,0..15] OF  TON;
	_arrTonOutput:		ARRAY[0..6,0..15] OF  TON;
	
	_arrFbMemory1:		ARRAY[0..6,0..15] OF FB_Memory1;
	
	_homeLineTon:		TON;// 线体正转延迟
	
	_fbPulse:			FB_Pulse;
	
	org:                 ARRAY[0..10] OF BOOL;
END_VAR

IF _bFirstRun THEN
	A_Info();
	_bFirstRun:=FALSE;
END_IF

A_InOut();// 输入输出
A_Axis();// 轴控制
A_Line();// 线体控制

IF GVL.stSetting.bDryRun THEN
	A_CylinderTest();
ELSE
	A_Cylinder();
END_IF

ACTION A_Axis:
FOR _i:=0 TO 20 BY 1 DO
	G_arrAxis[_i].ID:=TO_BYTE(_i+50);
END_FOR

org[_i]:=GVL_IO.arrAxisInput[_i].2;

_i:=E_Axis.TakeY;
IF GVL_Data.stRecipe.eMachineType=E_MachineType.RH311 OR GVL_Data.stRecipe.eMachineType=E_MachineType.LH311 THEN
    G_arrAxis[_i].stLock.bAll:=G_arrCylinder[E_Cylinder.TakeLift1].stOutput.bWork;
END_IF;
IF GVL_Data.stRecipe.eMachineType=E_MachineType.RH367 OR GVL_Data.stRecipe.eMachineType=E_MachineType.LH367 THEN
    G_arrAxis[_i].stLock.bAll:=G_arrCylinder[E_Cylinder.TakeLift1].stOutput.bWork AND G_arrCylinder[E_Cylinder.TakeLift2].stOutput.bWork;
END_IF;
G_arrAxisData[_i].stTorque.iGetTorque:=GVL_IO.arrGetTorque[_i];
GVL_IO.arrSetTorque[_i]:=TO_UINT(G_arrAxisData[_i].stTorque.iSetTorque);
G_arrAxisData[_i].stMode.iHomeMode:=0;
G_arrAxis[_i].stInput.bNegative:=GVL_IO.arrAxisInput[_i].0;
G_arrAxis[_i].stInput.bPositive:=GVL_IO.arrAxisInput[_i].2;

_i:=E_Axis.TakeZ;
G_arrAxis[_i].stLock.bShield:=GVL_Data.stRecipe.eMachineType=E_MachineType.LH311 OR GVL_Data.stRecipe.eMachineType=E_MachineType.RH311 OR GVL_Data.stRecipe.eMachineType=E_MachineType.RH367 OR  GVL_Data.stRecipe.eMachineType=E_MachineType.LH367; 
G_arrAxisData[_i].stTorque.iGetTorque:=GVL_IO.arrGetTorque[_i];
GVL_IO.arrSetTorque[_i]:=TO_UINT(G_arrAxisData[_i].stTorque.iSetTorque);
G_arrAxisData[_i].stMode.iHomeMode:=0;
G_arrAxis[_i].stInput.bNegative:=GVL_IO.arrAxisInput[_i].0;
G_arrAxis[_i].stInput.bPositive:=GVL_IO.arrAxisInput[_i].2;

_i:=E_Axis.UC_Y;
G_arrAxis[_i].stLock.bAll:=G_arrCylinder[E_Cylinder.UcLift].stOutput.bWork OR G_arrCylinder[E_Cylinder.UcSwing].stOutput.bWork;
G_arrAxis[_i].stLock.bShield:=GVL_Data.stRecipe.eMachineType<>E_MachineType.LH311 AND GVL_Data.stRecipe.eMachineType<>E_MachineType.RH311;
G_arrAxisData[_i].stTorque.iGetTorque:=GVL_IO.arrGetTorque[_i];
GVL_IO.arrSetTorque[_i]:=TO_UINT(G_arrAxisData[_i].stTorque.iSetTorque);
G_arrAxisData[_i].stMode.iHomeMode:=0;
G_arrAxis[_i].stInput.bNegative:=GVL_IO.arrAxisInput[_i].0;
G_arrAxis[_i].stInput.bPositive:=GVL_IO.arrAxisInput[_i].2;
END_ACTION

ACTION A_Cylinder:
FOR _i:=0 TO 50 BY 1 DO
	G_arrCylinder[_i].ID:=TO_BYTE(_i+50);
	G_arrCylinder[_i].stLock.bShield:=FALSE;
END_FOR


CASE GVL_Data.stRecipe.eMachineType OF
	E_MachineType.LH311,E_MachineType.RH311:
		G_arrCylinder[E_Cylinder.Line2OpenLateral2].stLock.bShield:=TRUE;
		G_arrCylinder[E_Cylinder.Line3OpenLateral2].stLock.bShield:=TRUE;
		G_arrCylinder[E_Cylinder.UcClamp1].stLock.bShield:=TRUE;
		G_arrCylinder[E_Cylinder.UcClamp2].stLock.bShield:=TRUE;
		G_arrCylinder[E_Cylinder.UcDrive].stLock.bShield:=TRUE;
		G_arrCylinder[E_Cylinder.UcLift1].stLock.bShield:=TRUE;
		G_arrCylinder[E_Cylinder.UcLift2].stLock.bShield:=TRUE;
		G_arrCylinder[E_Cylinder.UcRotate1].stLock.bShield:=TRUE;
		G_arrCylinder[E_Cylinder.UcRotate2].stLock.bShield:=TRUE;
	E_MachineType.LH353,E_MachineType.RH353:
		G_arrCylinder[E_Cylinder.Line2Standard2].stLock.bShield:=TRUE;
		G_arrCylinder[E_Cylinder.Line3Standard2].stLock.bShield:=TRUE;
		G_arrCylinder[E_Cylinder.TakeLift1].stLock.bShield:=TRUE;
		G_arrCylinder[E_Cylinder.TakeLift2].stLock.bShield:=TRUE;
		G_arrCylinder[E_Cylinder.UcClamp].stLock.bShield:=TRUE;
		G_arrCylinder[E_Cylinder.UcLift].stLock.bShield:=TRUE;
		G_arrCylinder[E_Cylinder.UcSwing].stLock.bShield:=TRUE;
	E_MachineType.LH367,E_MachineType.RH367:
		G_arrCylinder[E_Cylinder.Line2Standard2].stLock.bShield:=TRUE;
		G_arrCylinder[E_Cylinder.Line3Standard2].stLock.bShield:=TRUE;
		G_arrCylinder[E_Cylinder.UcClamp].stLock.bShield:=TRUE;
		G_arrCylinder[E_Cylinder.UcLift].stLock.bShield:=TRUE;
		G_arrCylinder[E_Cylinder.UcSwing].stLock.bShield:=TRUE;
	E_MachineType.LH201,E_MachineType.RH201:
		G_arrCylinder[E_Cylinder.Line2Standard1].stLock.bShield:=TRUE;
		G_arrCylinder[E_Cylinder.Line2Standard2].stLock.bShield:=TRUE;
		G_arrCylinder[E_Cylinder.Line3Standard1].stLock.bShield:=TRUE;
		G_arrCylinder[E_Cylinder.Line3Standard2].stLock.bShield:=TRUE;
		G_arrCylinder[E_Cylinder.TakeLift1].stLock.bShield:=TRUE;
		G_arrCylinder[E_Cylinder.TakeLift2].stLock.bShield:=TRUE;
		G_arrCylinder[E_Cylinder.UcClamp].stLock.bShield:=TRUE;
		G_arrCylinder[E_Cylinder.UcLift].stLock.bShield:=TRUE;
		G_arrCylinder[E_Cylinder.UcSwing].stLock.bShield:=TRUE;
	E_MachineType.LH069,E_MachineType.RH069:
		G_arrCylinder[E_Cylinder.Line2Standard1].stLock.bShield:=TRUE;
		G_arrCylinder[E_Cylinder.Line2Standard2].stLock.bShield:=TRUE;
		G_arrCylinder[E_Cylinder.Line3Standard1].stLock.bShield:=TRUE;
		G_arrCylinder[E_Cylinder.Line3Standard2].stLock.bShield:=TRUE;
		G_arrCylinder[E_Cylinder.TakeLift1].stLock.bShield:=TRUE;
		G_arrCylinder[E_Cylinder.TakeLift2].stLock.bShield:=TRUE;
		G_arrCylinder[E_Cylinder.UcClamp].stLock.bShield:=TRUE;
		G_arrCylinder[E_Cylinder.UcLift].stLock.bShield:=TRUE;
		G_arrCylinder[E_Cylinder.UcSwing].stLock.bShield:=TRUE;
	E_MachineType.LH373,E_MachineType.RH373:
		G_arrCylinder[E_Cylinder.Line2Standard2].stLock.bShield:=TRUE;
		G_arrCylinder[E_Cylinder.Line3Standard2].stLock.bShield:=TRUE;
		G_arrCylinder[E_Cylinder.Line2OpenLateral2].stLock.bShield:=TRUE;
		G_arrCylinder[E_Cylinder.Line3OpenLateral2].stLock.bShield:=TRUE;
		G_arrCylinder[E_Cylinder.TakeLift1].stLock.bShield:=TRUE;
		G_arrCylinder[E_Cylinder.TakeLift2].stLock.bShield:=TRUE;
		G_arrCylinder[E_Cylinder.UcClamp].stLock.bShield:=TRUE;
		G_arrCylinder[E_Cylinder.UcLift].stLock.bShield:=TRUE;
		G_arrCylinder[E_Cylinder.UcSwing].stLock.bShield:=TRUE;
END_CASE


_i:=E_Cylinder.Line0Part;
G_arrCylinder[_i].stInput.bHome:=GVL.I.bLine0Part_Cyl_H;
G_arrCylinder[_i].stInput.bWork:=GVL.I.bLine0Part_Cyl_W;
GVL.Q.bLine0Part_Cyl_H:=G_arrCylinder[_i].stOutput.bHome;
GVL.Q.bLine0Part_Cyl_W:=G_arrCylinder[_i].stOutput.bWork;

_i:=E_Cylinder.Line0Prevent;
G_arrCylinder[_i].stInput.bHome:=GVL.I.bLine0Prevent_Cyl_H;
G_arrCylinder[_i].stInput.bWork:=GVL.I.bLine0Prevent_Cyl_W;
GVL.Q.bLine0Prevent_Cyl_H:=G_arrCylinder[_i].stOutput.bHome;
GVL.Q.bLine0Prevent_Cyl_W:=G_arrCylinder[_i].stOutput.bWork;

_i:=E_Cylinder.Line1Elevator;
G_arrCylinder[_i].stInput.bHome:=NOT GVL.I.bLine1Elevator_Cyl_H;
G_arrCylinder[_i].stInput.bWork:=NOT GVL.I.bLine1Elevator_Cyl_W;
GVL.Q.bLine1Elevator_Cyl_H:=G_arrCylinder[_i].stOutput.bHome;
GVL.Q.bLine1Elevator_Cyl_W:=G_arrCylinder[_i].stOutput.bWork;

_i:=E_Cylinder.Line1Lift;
G_arrCylinder[_i].stInput.bHome:=GVL.I.bLine1Lift_Cyl_H;
G_arrCylinder[_i].stInput.bWork:=GVL.I.bLine1Lift_Cyl_W;
GVL.Q.bLine1Lift_Cyl_H:=G_arrCylinder[_i].stOutput.bHome;
GVL.Q.bLine1Lift_Cyl_W:=G_arrCylinder[_i].stOutput.bWork;

_i:=E_Cylinder.Line1Prevent;
G_arrCylinder[_i].stInput.bHome:=NOT G_arrCylinder[_i].stInput.bWork;
G_arrCylinder[_i].stInput.bWork:=GVL.I.bLine1Prevent_Cyl_W;
GVL.Q.bLine1Prevent_Cyl_H:=G_arrCylinder[_i].stOutput.bHome;
GVL.Q.bLine1Prevent_Cyl_W:=G_arrCylinder[_i].stOutput.bWork;

_i:=E_Cylinder.Line1Rotate;
G_arrCylinder[_i].stLock.bWork:=G_arrCylinder[E_Cylinder.Line1Lift].stOutput.bHome;
G_arrCylinder[_i].stLock.bHome:=G_arrCylinder[E_Cylinder.Line1Lift].stOutput.bHome;
G_arrCylinder[_i].stInput.bHome:=GVL.I.bLine1Rotate_Cyl_H;
G_arrCylinder[_i].stInput.bWork:=GVL.I.bLine1Rotate_Cyl_W;
GVL.Q.bLine1Rotate_Cyl_H:=G_arrCylinder[_i].stOutput.bHome;
GVL.Q.bLine1Rotate_Cyl_W:=G_arrCylinder[_i].stOutput.bWork;

_i:=E_Cylinder.Line1Adjust1;
G_arrCylinder[_i].stInput.bHome:=GVL.I.bLine1Adjust1_Cyl_H;
G_arrCylinder[_i].stInput.bWork:=GVL.I.bLine1Adjust1_Cyl_W;
GVL.Q.bLine1Adjust1_Cyl_H:=G_arrCylinder[_i].stOutput.bHome;
GVL.Q.bLine1Adjust1_Cyl_W:=G_arrCylinder[_i].stOutput.bWork;

_i:=E_Cylinder.Line2Lift;
G_arrCylinder[_i].stInput.bHome:=GVL.I.bLine2Lift_Cyl_H;
G_arrCylinder[_i].stInput.bWork:=GVL.I.bLine2Lift_Cyl_W;
GVL.Q.bLine2Lift_Cyl_H:=G_arrCylinder[_i].stOutput.bHome;
GVL.Q.bLine2Lift_Cyl_W:=G_arrCylinder[_i].stOutput.bWork;

_i:=E_Cylinder.Line2Prevent;
G_arrCylinder[_i].stInput.bHome:=NOT G_arrCylinder[_i].stInput.bWork;
G_arrCylinder[_i].stInput.bWork:=GVL.I.bLine2Prevent_Cyl_W;
GVL.Q.bLine2Prevent_Cyl_H:=G_arrCylinder[_i].stOutput.bHome;
GVL.Q.bLine2Prevent_Cyl_W:=G_arrCylinder[_i].stOutput.bWork;

_i:=E_Cylinder.Line2Standard1;
G_arrCylinder[_i].stInput.bHome:=GVL.I.bLine2Standard1_Cyl_H;
G_arrCylinder[_i].stInput.bWork:=GVL.I.bLine2Standard1_Cyl_W;
GVL.Q.bLine2Standard1_Cyl_H:=G_arrCylinder[_i].stOutput.bHome;
GVL.Q.bLine2Standard1_Cyl_W:=G_arrCylinder[_i].stOutput.bWork;

_i:=E_Cylinder.Line2Standard2;
G_arrCylinder[_i].stInput.bHome:=GVL.I.bLine2Standard2_Cyl_H;
G_arrCylinder[_i].stInput.bWork:=GVL.I.bLine2Standard2_Cyl_W;
GVL.Q.bLine2Standard2_Cyl_H:=G_arrCylinder[_i].stOutput.bHome;
GVL.Q.bLine2Standard2_Cyl_W:=G_arrCylinder[_i].stOutput.bWork;

_i:=E_Cylinder.Line2OpenLateral1;
G_arrCylinder[_i].stInput.bHome:=GVL.I.bLine2OpenLateral1_Cyl_H;
G_arrCylinder[_i].stInput.bWork:=GVL.I.bLine2OpenLateral1_Cyl_W;
GVL.Q.bLine2OpenLateral1_Cyl_H:=G_arrCylinder[_i].stOutput.bHome;
GVL.Q.bLine2OpenLateral1_Cyl_W:=G_arrCylinder[_i].stOutput.bWork;

_i:=E_Cylinder.Line2OpenRotate;
G_arrCylinder[_i].stLock.bHome:=G_arrCylinder[E_Cylinder.Line2OpenLateral2].stOutput.bWork;
G_arrCylinder[_i].stInput.bHome:=GVL.I.bLine2OpenRotate_Cyl_H;
G_arrCylinder[_i].stInput.bWork:=GVL.I.bLine2OpenRotate_Cyl_W;
GVL.Q.bLine2OpenRotate_Cyl_H:=G_arrCylinder[_i].stOutput.bHome;
GVL.Q.bLine2OpenRotate_Cyl_W:=G_arrCylinder[_i].stOutput.bWork;

_i:=E_Cylinder.Line2OpenLateral2;
G_arrCylinder[_i].stInput.bHome:=GVL.I.bLine2OpenLateral2_Cyl_H;
G_arrCylinder[_i].stInput.bWork:=G_arrCylinder[_i].stOutput.bWork;
GVL.Q.bLine2OpenLateral2_Cyl_H:=G_arrCylinder[_i].stOutput.bHome;
GVL.Q.bLine2OpenLateral2_Cyl_W:=G_arrCylinder[_i].stOutput.bWork;

_i:=E_Cylinder.Line3LoadLift;
G_arrCylinder[_i].stInput.bHome:=GVL.I.bLine3LoadLift_Cyl_H;
G_arrCylinder[_i].stInput.bWork:=GVL.I.bLine3LoadLift_Cyl_W;
GVL.Q.bLine3LoadLift_Cyl_H:=G_arrCylinder[_i].stOutput.bHome;
GVL.Q.bLine3LoadLift_Cyl_W:=G_arrCylinder[_i].stOutput.bWork;

_i:=E_Cylinder.Line3LoadPrevent;
G_arrCylinder[_i].stInput.bHome:=NOT G_arrCylinder[_i].stInput.bWork;
G_arrCylinder[_i].stInput.bWork:=GVL.I.bLine3LoadPrevent_Cyl_W;
GVL.Q.bLine3LoadPrevent_Cyl_H:=G_arrCylinder[_i].stOutput.bHome;
GVL.Q.bLine3LoadPrevent_Cyl_W:=G_arrCylinder[_i].stOutput.bWork;

_i:=E_Cylinder.Line3LoadRotate;
G_arrCylinder[_i].stLock.bWork:=G_arrCylinder[E_Cylinder.Line3LoadLift].stOutput.bHome;
G_arrCylinder[_i].stLock.bHome:=G_arrCylinder[E_Cylinder.Line3LoadLift].stOutput.bHome;
G_arrCylinder[_i].stInput.bHome:=GVL.I.bLine3LoadRotate_Cyl_H;
G_arrCylinder[_i].stInput.bWork:=GVL.I.bLine3LoadRotate_Cyl_W;
GVL.Q.bLine3LoadRotate_Cyl_H:=G_arrCylinder[_i].stOutput.bHome;
GVL.Q.bLine3LoadRotate_Cyl_W:=G_arrCylinder[_i].stOutput.bWork;

_i:=E_Cylinder.Line3OpenLift;
G_arrCylinder[_i].stInput.bHome:=GVL.I.bLine3OpenLift_Cyl_H;
G_arrCylinder[_i].stInput.bWork:=GVL.I.bLine3OpenLift_Cyl_W;
GVL.Q.bLine3OpenLift_Cyl_H:=G_arrCylinder[_i].stOutput.bHome;
GVL.Q.bLine3OpenLift_Cyl_W:=G_arrCylinder[_i].stOutput.bWork;

_i:=E_Cylinder.Line3OpenPrevent;
G_arrCylinder[_i].stInput.bHome:=NOT G_arrCylinder[_i].stInput.bWork;;
G_arrCylinder[_i].stInput.bWork:=GVL.I.bLine3OpenPrevent_Cyl_W;
GVL.Q.bLine3OpenPrevent_Cyl_H:=G_arrCylinder[_i].stOutput.bHome;
GVL.Q.bLine3OpenPrevent_Cyl_W:=G_arrCylinder[_i].stOutput.bWork;

_i:=E_Cylinder.Line3Standard1;
G_arrCylinder[_i].stInput.bHome:=GVL.I.bLine3Standard1_Cyl_H;
G_arrCylinder[_i].stInput.bWork:=GVL.I.bLine3Standard1_Cyl_W;
GVL.Q.bLine3Standard1_Cyl_H:=G_arrCylinder[_i].stOutput.bHome;
GVL.Q.bLine3Standard1_Cyl_W:=G_arrCylinder[_i].stOutput.bWork;

_i:=E_Cylinder.Line3Standard2;
G_arrCylinder[_i].stInput.bHome:=GVL.I.bLine3Standard2_Cyl_H;
G_arrCylinder[_i].stInput.bWork:=GVL.I.bLine3Standard2_Cyl_W;
GVL.Q.bLine3Standard2_Cyl_H:=G_arrCylinder[_i].stOutput.bHome;
GVL.Q.bLine3Standard2_Cyl_W:=G_arrCylinder[_i].stOutput.bWork;

_i:=E_Cylinder.Line3OpenLateral1;
G_arrCylinder[_i].stInput.bHome:=GVL.I.bLine3OpenLateral1_Cyl_H;
G_arrCylinder[_i].stInput.bWork:=GVL.I.bLine3OpenLateral1_Cyl_W;
GVL.Q.bLine3OpenLateral1_Cyl_H:=G_arrCylinder[_i].stOutput.bHome;
GVL.Q.bLine3OpenLateral1_Cyl_W:=G_arrCylinder[_i].stOutput.bWork;

_i:=E_Cylinder.Line3OpenRotate;
G_arrCylinder[_i].stLock.bHome:=G_arrCylinder[E_Cylinder.Line3OpenLateral2].stOutput.bWork;
G_arrCylinder[_i].stInput.bHome:=GVL.I.bLine3OpenRotate_Cyl_H;
G_arrCylinder[_i].stInput.bWork:=GVL.I.bLine3OpenRotate_Cyl_W;
GVL.Q.bLine3OpenRotate_Cyl_H:=G_arrCylinder[_i].stOutput.bHome;
GVL.Q.bLine3OpenRotate_Cyl_W:=G_arrCylinder[_i].stOutput.bWork;

_i:=E_Cylinder.Line3OpenLateral2;
G_arrCylinder[_i].stInput.bHome:=GVL.I.bLine3OpenLateral2_Cyl_H;
G_arrCylinder[_i].stInput.bWork:=G_arrCylinder[_i].stOutput.bWork;
GVL.Q.bLine3OpenLateral2_Cyl_H:=G_arrCylinder[_i].stOutput.bHome;
GVL.Q.bLine3OpenLateral2_Cyl_W:=G_arrCylinder[_i].stOutput.bWork;

_i:=E_Cylinder.TakeLift1;
G_arrCylinder[_i].stInput.bHome:=GVL.I.bTakeLift1_Cyl_H;
G_arrCylinder[_i].stInput.bWork:=GVL.I.bTakeLift1_Cyl_W;
GVL.Q.bTakeLift1_Cyl_H:=G_arrCylinder[_i].stOutput.bHome;
GVL.Q.bTakeLift1_Cyl_W:=G_arrCylinder[_i].stOutput.bWork;

_i:=E_Cylinder.TakeLift2;
G_arrCylinder[_i].stInput.bHome:=GVL.I.bTakeLift2_Cyl_H;
G_arrCylinder[_i].stInput.bWork:=GVL.I.bTakeLift2_Cyl_W;
GVL.Q.bTakeLift2_Cyl_H:=G_arrCylinder[_i].stOutput.bHome;
GVL.Q.bTakeLift2_Cyl_W:=G_arrCylinder[_i].stOutput.bWork;

_i:=E_Cylinder.TakeClamp;
G_arrCylinder[_i].stInput.bHome:=GVL.I.bTakeClamp_Cyl_H;
G_arrCylinder[_i].stInput.bWork:=GVL.I.bTakeClamp_Cyl_W;
GVL.Q.bTakeClamp_Cyl_H:=G_arrCylinder[_i].stOutput.bHome;
GVL.Q.bTakeClamp_Cyl_W:=G_arrCylinder[_i].stOutput.bWork;

_i:=E_Cylinder.UcLift;
G_arrCylinder[_i].stInput.bHome:=GVL.I.bUcLift_Cyl_H;
G_arrCylinder[_i].stInput.bWork:=GVL.I.bUcLift_Cyl_W;
GVL.Q.bUcLift_Cyl_H:=G_arrCylinder[_i].stOutput.bHome;
GVL.Q.bUcLift_Cyl_W:=G_arrCylinder[_i].stOutput.bWork;

_i:=E_Cylinder.UcClamp;
G_arrCylinder[_i].stInput.bHome:=GVL.I.bUcClamp_Cyl_H;
G_arrCylinder[_i].stInput.bWork:=GVL.I.bUcClamp_Cyl_W;
GVL.Q.bUcClamp_Cyl_H:=G_arrCylinder[_i].stOutput.bHome;
GVL.Q.bUcClamp_Cyl_W:=G_arrCylinder[_i].stOutput.bWork;

_i:=E_Cylinder.UcSwing;
G_arrCylinder[_i].stInput.bHome:=GVL.I.bUcSwing_Cyl_H;
G_arrCylinder[_i].stInput.bWork:=GVL.I.bUcSwing_Cyl_W;
GVL.Q.bUcSwing_Cyl_H:=G_arrCylinder[_i].stOutput.bHome;
GVL.Q.bUcSwing_Cyl_W:=G_arrCylinder[_i].stOutput.bWork;

_i:=E_Cylinder.UcLift1;
G_arrCylinder[_i].stLock.bHome:=G_arrCylinder[E_Cylinder.UcRotate1].stOutput.bWork OR G_arrCylinder[E_Cylinder.Line2OpenLateral2].stOutput.bWork;
G_arrCylinder[_i].stLock.bWork:=G_arrCylinder[E_Cylinder.UcRotate1].stOutput.bWork OR G_arrCylinder[E_Cylinder.Line2OpenLateral2].stOutput.bWork;
G_arrCylinder[_i].stInput.bHome:=GVL.I.bUcLift1_Cyl_H;
G_arrCylinder[_i].stInput.bWork:=GVL.I.bUcLift1_Cyl_W;
GVL.Q.bUcLift1_Cyl_H:=G_arrCylinder[_i].stOutput.bHome;
GVL.Q.bUcLift1_Cyl_W:=G_arrCylinder[_i].stOutput.bWork;

_i:=E_Cylinder.UcClamp1;
G_arrCylinder[_i].stInput.bHome:=GVL.I.bUcClamp1_Cyl_H;
G_arrCylinder[_i].stInput.bWork:=GVL.I.bUcClamp1_Cyl_W;
GVL.Q.bUcClamp1_Cyl_H:=G_arrCylinder[_i].stOutput.bHome;
GVL.Q.bUcClamp1_Cyl_W:=G_arrCylinder[_i].stOutput.bWork;

_i:=E_Cylinder.UcRotate1;
G_arrCylinder[_i].stLock.bHome:=G_arrCylinder[E_Cylinder.UcLift1].stOutput.bHome ;
G_arrCylinder[_i].stLock.bWork:=G_arrCylinder[E_Cylinder.UcLift1].stOutput.bHome ;
G_arrCylinder[_i].stInput.bHome:=GVL.I.bUcRotate1_Cyl_H;
G_arrCylinder[_i].stInput.bWork:=GVL.I.bUcRotate1_Cyl_W;
GVL.Q.bUcRotate1_Cyl_H:=G_arrCylinder[_i].stOutput.bHome;
GVL.Q.bUcRotate1_Cyl_W:=G_arrCylinder[_i].stOutput.bWork;

_i:=E_Cylinder.UcLift2;
G_arrCylinder[_i].stLock.bHome:=G_arrCylinder[E_Cylinder.UcRotate2].stOutput.bWork OR G_arrCylinder[E_Cylinder.Line3OpenLateral2].stOutput.bWork;
G_arrCylinder[_i].stLock.bWork:=G_arrCylinder[E_Cylinder.UcRotate2].stOutput.bWork OR G_arrCylinder[E_Cylinder.Line3OpenLateral2].stOutput.bWork;
G_arrCylinder[_i].stInput.bHome:=GVL.I.bUcLift2_Cyl_H;
G_arrCylinder[_i].stInput.bWork:=GVL.I.bUcLift2_Cyl_W;
GVL.Q.bUcLift2_Cyl_H:=G_arrCylinder[_i].stOutput.bHome;
GVL.Q.bUcLift2_Cyl_W:=G_arrCylinder[_i].stOutput.bWork;

_i:=E_Cylinder.UcClamp2;
G_arrCylinder[_i].stInput.bHome:=GVL.I.bUcClamp2_Cyl_H;
G_arrCylinder[_i].stInput.bWork:=GVL.I.bUcClamp2_Cyl_W;
GVL.Q.bUcClamp2_Cyl_H:=G_arrCylinder[_i].stOutput.bHome;
GVL.Q.bUcClamp2_Cyl_W:=G_arrCylinder[_i].stOutput.bWork;

_i:=E_Cylinder.UcRotate2;
G_arrCylinder[_i].stLock.bHome:=G_arrCylinder[E_Cylinder.UcLift2].stOutput.bHome;
G_arrCylinder[_i].stLock.bWork:=G_arrCylinder[E_Cylinder.UcLift2].stOutput.bHome;
G_arrCylinder[_i].stInput.bHome:=GVL.I.bUcRotate2_Cyl_H;
G_arrCylinder[_i].stInput.bWork:=GVL.I.bUcRotate2_Cyl_W;
GVL.Q.bUcRotate2_Cyl_H:=G_arrCylinder[_i].stOutput.bHome;
GVL.Q.bUcRotate2_Cyl_W:=G_arrCylinder[_i].stOutput.bWork;

_i:=E_Cylinder.UcDrive;
G_arrCylinder[_i].stInput.bHome:=GVL.I.bUcDrive_Cyl_H;
G_arrCylinder[_i].stInput.bWork:=GVL.I.bUcDrive_Cyl_W;
GVL.Q.bUcDrive_Cyl_H:=G_arrCylinder[_i].stOutput.bHome;
GVL.Q.bUcDrive_Cyl_W:=G_arrCylinder[_i].stOutput.bWork;

_i:=E_Cylinder.FrockElevator1;
G_arrCylinder[_i].stInput.bHome:=NOT  GVL.I.bFrockElevator1_Cyl_H;
G_arrCylinder[_i].stInput.bWork:=NOT  GVL.I.bFrockElevator1_Cyl_W;
GVL.Q.bFrockElevator1_Cyl_H:=G_arrCylinder[_i].stOutput.bHome;
GVL.Q.bFrockElevator1_Cyl_W:=G_arrCylinder[_i].stOutput.bWork;

_i:=E_Cylinder.FrockRotateDown1;
G_arrCylinder[_i].stInput.bHome:=NOT  GVL.I.bFrockRotateDown1_Cyl_W;
G_arrCylinder[_i].stInput.bWork:=GVL.I.bFrockRotateDown1_Cyl_W;
GVL.Q.bFrockRotateDown1_Cyl_H:=G_arrCylinder[_i].stOutput.bHome;
GVL.Q.bFrockRotateDown1_Cyl_W:=G_arrCylinder[_i].stOutput.bWork;

_i:=E_Cylinder.FrockPush1;
G_arrCylinder[_i].stInput.bHome:=GVL.I.bFrockPush1_Cyl_H;
G_arrCylinder[_i].stInput.bWork:=GVL.I.bFrockPush1_Cyl_W;
GVL.Q.bFrockPush1_Cyl_H:=G_arrCylinder[_i].stOutput.bHome;
GVL.Q.bFrockPush1_Cyl_W:=G_arrCylinder[_i].stOutput.bWork;

_i:=E_Cylinder.FrockElevator2;
G_arrCylinder[_i].stInput.bHome:=NOT  GVL.I.bFrockElevator2_Cyl_H;
G_arrCylinder[_i].stInput.bWork:=NOT  GVL.I.bFrockElevator2_Cyl_W;
GVL.Q.bFrockElevator2_Cyl_H:=G_arrCylinder[_i].stOutput.bHome;
GVL.Q.bFrockElevator2_Cyl_W:=G_arrCylinder[_i].stOutput.bWork;

_i:=E_Cylinder.FrockRotateDown2;
G_arrCylinder[_i].stInput.bHome:=NOT GVL.I.bFrockRotateDown2_Cyl_W;
G_arrCylinder[_i].stInput.bWork:=GVL.I.bFrockRotateDown2_Cyl_W;
GVL.Q.bFrockRotateDown2_Cyl_H:=G_arrCylinder[_i].stOutput.bHome;
GVL.Q.bFrockRotateDown2_Cyl_W:=G_arrCylinder[_i].stOutput.bWork;

_i:=E_Cylinder.FrockPush2;
G_arrCylinder[_i].stInput.bHome:=GVL.I.bFrockPush2_Cyl_H;
G_arrCylinder[_i].stInput.bWork:=GVL.I.bFrockPush2_Cyl_W;
GVL.Q.bFrockPush2_Cyl_H:=G_arrCylinder[_i].stOutput.bHome;
GVL.Q.bFrockPush2_Cyl_W:=G_arrCylinder[_i].stOutput.bWork;

_i:=E_Cylinder.FrockBelt;
G_arrCylinder[_i].stInput.bHome:=GVL.I.bFrockBelt_Cyl_H;
G_arrCylinder[_i].stInput.bWork:=GVL.I.bFrockBelt_Cyl_W;
GVL.Q.bFrockBelt_Cyl_H:=G_arrCylinder[_i].stOutput.bHome;
GVL.Q.bFrockBelt_Cyl_W:=G_arrCylinder[_i].stOutput.bWork;
END_ACTION

ACTION A_CylinderTest:
FOR _i:=0 TO 50 BY 1 DO
	G_arrCylinder[_i].ID:=TO_BYTE(_i+50);
	_arrCylTon_H[_i](IN:=G_arrCylinder[_i].stOutput.bHome , PT:=T#2S , Q=> , ET=> );
	_arrCylTon_W[_i](IN:=G_arrCylinder[_i].stOutput.bWork , PT:=T#2S , Q=> , ET=> );
	G_arrCylinder[_i].stInput.bHome:=_arrCylTon_H[_i].Q;
	G_arrCylinder[_i].stInput.bWork:=_arrCylTon_W[_i].Q;
END_FOR

FOR _i:=0 TO 50 BY 1 DO
	G_arrCylinder[_i].ID:=TO_BYTE(_i+50);
	G_arrCylinder[_i].stLock.bShield:=FALSE;
END_FOR


CASE GVL_Data.stRecipe.eMachineType OF
	E_MachineType.LH311,E_MachineType.RH311:
		G_arrCylinder[E_Cylinder.Line2OpenLateral2].stLock.bShield:=TRUE;
		G_arrCylinder[E_Cylinder.Line3OpenLateral2].stLock.bShield:=TRUE;
		G_arrCylinder[E_Cylinder.UcClamp1].stLock.bShield:=TRUE;
		G_arrCylinder[E_Cylinder.UcClamp2].stLock.bShield:=TRUE;
		G_arrCylinder[E_Cylinder.UcDrive].stLock.bShield:=TRUE;
		G_arrCylinder[E_Cylinder.UcLift1].stLock.bShield:=TRUE;
		G_arrCylinder[E_Cylinder.UcLift2].stLock.bShield:=TRUE;
		G_arrCylinder[E_Cylinder.UcRotate1].stLock.bShield:=TRUE;
		G_arrCylinder[E_Cylinder.UcRotate2].stLock.bShield:=TRUE;
	E_MachineType.LH353,E_MachineType.RH353:
		G_arrCylinder[E_Cylinder.Line2Standard2].stLock.bShield:=TRUE;
		G_arrCylinder[E_Cylinder.Line3Standard2].stLock.bShield:=TRUE;
		G_arrCylinder[E_Cylinder.TakeLift1].stLock.bShield:=TRUE;
		G_arrCylinder[E_Cylinder.TakeLift2].stLock.bShield:=TRUE;
		G_arrCylinder[E_Cylinder.UcClamp].stLock.bShield:=TRUE;
		G_arrCylinder[E_Cylinder.UcLift].stLock.bShield:=TRUE;
		G_arrCylinder[E_Cylinder.UcSwing].stLock.bShield:=TRUE;
	E_MachineType.LH367,E_MachineType.RH367:
		G_arrCylinder[E_Cylinder.Line2Standard2].stLock.bShield:=TRUE;
		G_arrCylinder[E_Cylinder.Line3Standard2].stLock.bShield:=TRUE;
		G_arrCylinder[E_Cylinder.UcClamp].stLock.bShield:=TRUE;
		G_arrCylinder[E_Cylinder.UcLift].stLock.bShield:=TRUE;
		G_arrCylinder[E_Cylinder.UcSwing].stLock.bShield:=TRUE;
	E_MachineType.LH201,E_MachineType.RH201:
		G_arrCylinder[E_Cylinder.Line2Standard1].stLock.bShield:=TRUE;
		G_arrCylinder[E_Cylinder.Line2Standard2].stLock.bShield:=TRUE;
		G_arrCylinder[E_Cylinder.Line3Standard1].stLock.bShield:=TRUE;
		G_arrCylinder[E_Cylinder.Line3Standard2].stLock.bShield:=TRUE;
		G_arrCylinder[E_Cylinder.TakeLift1].stLock.bShield:=TRUE;
		G_arrCylinder[E_Cylinder.TakeLift2].stLock.bShield:=TRUE;
		G_arrCylinder[E_Cylinder.UcClamp].stLock.bShield:=TRUE;
		G_arrCylinder[E_Cylinder.UcLift].stLock.bShield:=TRUE;
		G_arrCylinder[E_Cylinder.UcSwing].stLock.bShield:=TRUE;
	E_MachineType.LH069,E_MachineType.RH069:
		G_arrCylinder[E_Cylinder.Line2Standard1].stLock.bShield:=TRUE;
		G_arrCylinder[E_Cylinder.Line2Standard2].stLock.bShield:=TRUE;
		G_arrCylinder[E_Cylinder.Line3Standard1].stLock.bShield:=TRUE;
		G_arrCylinder[E_Cylinder.Line3Standard2].stLock.bShield:=TRUE;
		G_arrCylinder[E_Cylinder.TakeLift1].stLock.bShield:=TRUE;
		G_arrCylinder[E_Cylinder.TakeLift2].stLock.bShield:=TRUE;
		G_arrCylinder[E_Cylinder.UcClamp].stLock.bShield:=TRUE;
		G_arrCylinder[E_Cylinder.UcLift].stLock.bShield:=TRUE;
		G_arrCylinder[E_Cylinder.UcSwing].stLock.bShield:=TRUE;
	E_MachineType.LH373,E_MachineType.RH373:
		G_arrCylinder[E_Cylinder.Line2Standard2].stLock.bShield:=TRUE;
		G_arrCylinder[E_Cylinder.Line3Standard2].stLock.bShield:=TRUE;
		G_arrCylinder[E_Cylinder.Line2OpenLateral2].stLock.bShield:=TRUE;
		G_arrCylinder[E_Cylinder.Line3OpenLateral2].stLock.bShield:=TRUE;
		G_arrCylinder[E_Cylinder.TakeLift1].stLock.bShield:=TRUE;
		G_arrCylinder[E_Cylinder.TakeLift2].stLock.bShield:=TRUE;
		G_arrCylinder[E_Cylinder.UcClamp].stLock.bShield:=TRUE;
		G_arrCylinder[E_Cylinder.UcLift].stLock.bShield:=TRUE;
		G_arrCylinder[E_Cylinder.UcSwing].stLock.bShield:=TRUE;
END_CASE


_i:=E_Cylinder.Line0Part;
GVL.Q.bLine0Part_Cyl_H:=G_arrCylinder[_i].stOutput.bHome;
GVL.Q.bLine0Part_Cyl_W:=G_arrCylinder[_i].stOutput.bWork;

_i:=E_Cylinder.Line0Prevent;
GVL.Q.bLine0Prevent_Cyl_H:=G_arrCylinder[_i].stOutput.bHome;
GVL.Q.bLine0Prevent_Cyl_W:=G_arrCylinder[_i].stOutput.bWork;

_i:=E_Cylinder.Line1Elevator;
GVL.Q.bLine1Elevator_Cyl_H:=G_arrCylinder[_i].stOutput.bHome;
GVL.Q.bLine1Elevator_Cyl_W:=G_arrCylinder[_i].stOutput.bWork;

_i:=E_Cylinder.Line1Lift;
GVL.Q.bLine1Lift_Cyl_H:=G_arrCylinder[_i].stOutput.bHome;
GVL.Q.bLine1Lift_Cyl_W:=G_arrCylinder[_i].stOutput.bWork;

_i:=E_Cylinder.Line1Prevent;
GVL.Q.bLine1Prevent_Cyl_H:=G_arrCylinder[_i].stOutput.bHome;
GVL.Q.bLine1Prevent_Cyl_W:=G_arrCylinder[_i].stOutput.bWork;

_i:=E_Cylinder.Line1Rotate;
GVL.Q.bLine1Rotate_Cyl_H:=G_arrCylinder[_i].stOutput.bHome;
GVL.Q.bLine1Rotate_Cyl_W:=G_arrCylinder[_i].stOutput.bWork;

_i:=E_Cylinder.Line1Adjust1;
GVL.Q.bLine1Adjust1_Cyl_H:=G_arrCylinder[_i].stOutput.bHome;
GVL.Q.bLine1Adjust1_Cyl_W:=G_arrCylinder[_i].stOutput.bWork;

_i:=E_Cylinder.Line2Lift;
GVL.Q.bLine2Lift_Cyl_H:=G_arrCylinder[_i].stOutput.bHome;
GVL.Q.bLine2Lift_Cyl_W:=G_arrCylinder[_i].stOutput.bWork;

_i:=E_Cylinder.Line2Prevent;
GVL.Q.bLine2Prevent_Cyl_H:=G_arrCylinder[_i].stOutput.bHome;
GVL.Q.bLine2Prevent_Cyl_W:=G_arrCylinder[_i].stOutput.bWork;

_i:=E_Cylinder.Line2Standard1;
GVL.Q.bLine2Standard1_Cyl_H:=G_arrCylinder[_i].stOutput.bHome;
GVL.Q.bLine2Standard1_Cyl_W:=G_arrCylinder[_i].stOutput.bWork;

_i:=E_Cylinder.Line2Standard2;
GVL.Q.bLine2Standard2_Cyl_H:=G_arrCylinder[_i].stOutput.bHome;
GVL.Q.bLine2Standard2_Cyl_W:=G_arrCylinder[_i].stOutput.bWork;

_i:=E_Cylinder.Line2OpenLateral1;
GVL.Q.bLine2OpenLateral1_Cyl_H:=G_arrCylinder[_i].stOutput.bHome;
GVL.Q.bLine2OpenLateral1_Cyl_W:=G_arrCylinder[_i].stOutput.bWork;

_i:=E_Cylinder.Line2OpenRotate;
GVL.Q.bLine2OpenRotate_Cyl_H:=G_arrCylinder[_i].stOutput.bHome;
GVL.Q.bLine2OpenRotate_Cyl_W:=G_arrCylinder[_i].stOutput.bWork;

_i:=E_Cylinder.Line2OpenLateral2;
GVL.Q.bLine2OpenLateral2_Cyl_H:=G_arrCylinder[_i].stOutput.bHome;
GVL.Q.bLine2OpenLateral2_Cyl_W:=G_arrCylinder[_i].stOutput.bWork;

_i:=E_Cylinder.Line3LoadLift;
GVL.Q.bLine3LoadLift_Cyl_H:=G_arrCylinder[_i].stOutput.bHome;
GVL.Q.bLine3LoadLift_Cyl_W:=G_arrCylinder[_i].stOutput.bWork;

_i:=E_Cylinder.Line3LoadPrevent;
GVL.Q.bLine3LoadPrevent_Cyl_H:=G_arrCylinder[_i].stOutput.bHome;
GVL.Q.bLine3LoadPrevent_Cyl_W:=G_arrCylinder[_i].stOutput.bWork;

_i:=E_Cylinder.Line3LoadRotate;
GVL.Q.bLine3LoadRotate_Cyl_H:=G_arrCylinder[_i].stOutput.bHome;
GVL.Q.bLine3LoadRotate_Cyl_W:=G_arrCylinder[_i].stOutput.bWork;

_i:=E_Cylinder.Line3OpenLift;
GVL.Q.bLine3OpenLift_Cyl_H:=G_arrCylinder[_i].stOutput.bHome;
GVL.Q.bLine3OpenLift_Cyl_W:=G_arrCylinder[_i].stOutput.bWork;

_i:=E_Cylinder.Line3OpenPrevent;
GVL.Q.bLine3OpenPrevent_Cyl_H:=G_arrCylinder[_i].stOutput.bHome;
GVL.Q.bLine3OpenPrevent_Cyl_W:=G_arrCylinder[_i].stOutput.bWork;

_i:=E_Cylinder.Line3Standard1;
GVL.Q.bLine3Standard1_Cyl_H:=G_arrCylinder[_i].stOutput.bHome;
GVL.Q.bLine3Standard1_Cyl_W:=G_arrCylinder[_i].stOutput.bWork;

_i:=E_Cylinder.Line3Standard2;
GVL.Q.bLine3Standard2_Cyl_H:=G_arrCylinder[_i].stOutput.bHome;
GVL.Q.bLine3Standard2_Cyl_W:=G_arrCylinder[_i].stOutput.bWork;

_i:=E_Cylinder.Line3OpenLateral1;
GVL.Q.bLine3OpenLateral1_Cyl_H:=G_arrCylinder[_i].stOutput.bHome;
GVL.Q.bLine3OpenLateral1_Cyl_W:=G_arrCylinder[_i].stOutput.bWork;

_i:=E_Cylinder.Line3OpenRotate;
GVL.Q.bLine3OpenRotate_Cyl_H:=G_arrCylinder[_i].stOutput.bHome;
GVL.Q.bLine3OpenRotate_Cyl_W:=G_arrCylinder[_i].stOutput.bWork;

_i:=E_Cylinder.Line3OpenLateral2;
GVL.Q.bLine3OpenLateral2_Cyl_H:=G_arrCylinder[_i].stOutput.bHome;
GVL.Q.bLine3OpenLateral2_Cyl_W:=G_arrCylinder[_i].stOutput.bWork;

_i:=E_Cylinder.TakeLift1;
GVL.Q.bTakeLift1_Cyl_H:=G_arrCylinder[_i].stOutput.bHome;
GVL.Q.bTakeLift1_Cyl_W:=G_arrCylinder[_i].stOutput.bWork;

_i:=E_Cylinder.TakeLift2;
GVL.Q.bTakeLift2_Cyl_H:=G_arrCylinder[_i].stOutput.bHome;
GVL.Q.bTakeLift2_Cyl_W:=G_arrCylinder[_i].stOutput.bWork;

_i:=E_Cylinder.TakeClamp;
GVL.Q.bTakeClamp_Cyl_H:=G_arrCylinder[_i].stOutput.bHome;
GVL.Q.bTakeClamp_Cyl_W:=G_arrCylinder[_i].stOutput.bWork;

_i:=E_Cylinder.UcLift;
GVL.Q.bUcLift_Cyl_H:=G_arrCylinder[_i].stOutput.bHome;
GVL.Q.bUcLift_Cyl_W:=G_arrCylinder[_i].stOutput.bWork;

_i:=E_Cylinder.UcClamp;
GVL.Q.bUcClamp_Cyl_H:=G_arrCylinder[_i].stOutput.bHome;
GVL.Q.bUcClamp_Cyl_W:=G_arrCylinder[_i].stOutput.bWork;

_i:=E_Cylinder.UcSwing;
GVL.Q.bUcSwing_Cyl_H:=G_arrCylinder[_i].stOutput.bHome;
GVL.Q.bUcSwing_Cyl_W:=G_arrCylinder[_i].stOutput.bWork;

_i:=E_Cylinder.UcLift1;
GVL.Q.bUcLift1_Cyl_H:=G_arrCylinder[_i].stOutput.bHome;
GVL.Q.bUcLift1_Cyl_W:=G_arrCylinder[_i].stOutput.bWork;

_i:=E_Cylinder.UcClamp1;
GVL.Q.bUcClamp1_Cyl_H:=G_arrCylinder[_i].stOutput.bHome;
GVL.Q.bUcClamp1_Cyl_W:=G_arrCylinder[_i].stOutput.bWork;

_i:=E_Cylinder.UcRotate1;
GVL.Q.bUcRotate1_Cyl_H:=G_arrCylinder[_i].stOutput.bHome;
GVL.Q.bUcRotate1_Cyl_W:=G_arrCylinder[_i].stOutput.bWork;

_i:=E_Cylinder.UcLift2;
GVL.Q.bUcLift2_Cyl_H:=G_arrCylinder[_i].stOutput.bHome;
GVL.Q.bUcLift2_Cyl_W:=G_arrCylinder[_i].stOutput.bWork;

_i:=E_Cylinder.UcClamp2;
GVL.Q.bUcClamp2_Cyl_H:=G_arrCylinder[_i].stOutput.bHome;
GVL.Q.bUcClamp2_Cyl_W:=G_arrCylinder[_i].stOutput.bWork;

_i:=E_Cylinder.UcRotate2;
GVL.Q.bUcRotate2_Cyl_H:=G_arrCylinder[_i].stOutput.bHome;
GVL.Q.bUcRotate2_Cyl_W:=G_arrCylinder[_i].stOutput.bWork;

_i:=E_Cylinder.UcDrive;
GVL.Q.bUcDrive_Cyl_H:=G_arrCylinder[_i].stOutput.bHome;
GVL.Q.bUcDrive_Cyl_W:=G_arrCylinder[_i].stOutput.bWork;

_i:=E_Cylinder.FrockElevator1;
GVL.Q.bFrockElevator1_Cyl_H:=G_arrCylinder[_i].stOutput.bHome;
GVL.Q.bFrockElevator1_Cyl_W:=G_arrCylinder[_i].stOutput.bWork;

_i:=E_Cylinder.FrockRotateDown1;
GVL.Q.bFrockRotateDown1_Cyl_H:=G_arrCylinder[_i].stOutput.bHome;
GVL.Q.bFrockRotateDown1_Cyl_W:=G_arrCylinder[_i].stOutput.bWork;

_i:=E_Cylinder.FrockPush1;
GVL.Q.bFrockPush1_Cyl_H:=G_arrCylinder[_i].stOutput.bHome;
GVL.Q.bFrockPush1_Cyl_W:=G_arrCylinder[_i].stOutput.bWork;

_i:=E_Cylinder.FrockElevator2;
GVL.Q.bFrockElevator2_Cyl_H:=G_arrCylinder[_i].stOutput.bHome;
GVL.Q.bFrockElevator2_Cyl_W:=G_arrCylinder[_i].stOutput.bWork;

_i:=E_Cylinder.FrockRotateDown2;
GVL.Q.bFrockRotateDown2_Cyl_H:=G_arrCylinder[_i].stOutput.bHome;
GVL.Q.bFrockRotateDown2_Cyl_W:=G_arrCylinder[_i].stOutput.bWork;

_i:=E_Cylinder.FrockPush2;
GVL.Q.bFrockPush2_Cyl_H:=G_arrCylinder[_i].stOutput.bHome;
GVL.Q.bFrockPush2_Cyl_W:=G_arrCylinder[_i].stOutput.bWork;

_i:=E_Cylinder.FrockBelt;
GVL.Q.bFrockBelt_Cyl_H:=G_arrCylinder[_i].stOutput.bHome;
GVL.Q.bFrockBelt_Cyl_W:=G_arrCylinder[_i].stOutput.bWork;
END_ACTION

ACTION A_Info:
_i:=E_Axis.TakeY;
G_arrAxis[_i].arrInfo[E_Language.Chinese].sName:="取料Y轴";
G_arrAxis[_i].arrInfo[E_Language.English].sName:="TakeY";
G_arrAxis[_i].arrInfo[E_Language.Vietnamese].sName:="Lấy vật liệu trên trục Y";

_i:=E_Axis.TakeZ;
G_arrAxis[_i].arrInfo[E_Language.Chinese].sName:="取料Z轴";
G_arrAxis[_i].arrInfo[E_Language.English].sName:="TakeZ";
G_arrAxis[_i].arrInfo[E_Language.Vietnamese].sName:="Lấy trục Z";

_i:=E_Axis.UC_Y;
G_arrAxis[_i].arrInfo[E_Language.Chinese].sName:="下UC_Y轴";
G_arrAxis[_i].arrInfo[E_Language.English].sName:="UC_Y";
G_arrAxis[_i].arrInfo[E_Language.Vietnamese].sName:="Trục dưới UC_Y";

_i:=E_Cylinder.Line0Part;
G_arrCylinder[_i].arrInfo[E_Language.Chinese].sName:="主流线分料气缸";
G_arrCylinder[_i].arrInfo[E_Language.English].sName:="Line0Part";
G_arrCylinder[_i].arrInfo[E_Language.Vietnamese].sName:="Xi lanh phân phối dòng chính";

_i:=E_Cylinder.Line0Prevent;
G_arrCylinder[_i].arrInfo[E_Language.Chinese].sName:="主流线阻挡气缸";
G_arrCylinder[_i].arrInfo[E_Language.English].sName:="Line0Prevent";
G_arrCylinder[_i].arrInfo[E_Language.Vietnamese].sName:="Dòng chính ngăn chặn các xi lanh";

_i:=E_Cylinder.Line1Elevator;
G_arrCylinder[_i].arrInfo[E_Language.Chinese].sName:="流水线1提升气缸";
G_arrCylinder[_i].arrInfo[E_Language.English].sName:="Line1Elevator";
G_arrCylinder[_i].arrInfo[E_Language.Vietnamese].sName:="Xi lanh nâng cấp dòng 1";

_i:=E_Cylinder.Line1Lift;
G_arrCylinder[_i].arrInfo[E_Language.Chinese].sName:="流水线1顶升气缸";
G_arrCylinder[_i].arrInfo[E_Language.English].sName:="Line1Lift";
G_arrCylinder[_i].arrInfo[E_Language.Vietnamese].sName:="Xi lanh 1 lít đường ống";

_i:=E_Cylinder.Line1Prevent;
G_arrCylinder[_i].arrInfo[E_Language.Chinese].sName:="流水线1阻挡气缸";
G_arrCylinder[_i].arrInfo[E_Language.English].sName:="Line1Prevent";
G_arrCylinder[_i].arrInfo[E_Language.Vietnamese].sName:="Xi lanh chặn đường ống 1";

_i:=E_Cylinder.Line1Rotate;
G_arrCylinder[_i].arrInfo[E_Language.Chinese].sName:="流水线1旋转气缸";
G_arrCylinder[_i].arrInfo[E_Language.English].sName:="Line1Rotate";
G_arrCylinder[_i].arrInfo[E_Language.Vietnamese].sName:="Xi lanh xoay dòng 1";

_i:=E_Cylinder.Line1Adjust1;
G_arrCylinder[_i].arrInfo[E_Language.Chinese].sName:="流水线1调宽气缸1";
G_arrCylinder[_i].arrInfo[E_Language.English].sName:="Line1Adjust1";
G_arrCylinder[_i].arrInfo[E_Language.Vietnamese].sName:="Đường ống 1 mở rộng xi lanh 1";

_i:=E_Cylinder.Line2Lift;
G_arrCylinder[_i].arrInfo[E_Language.Chinese].sName:="流水线2顶升气缸";
G_arrCylinder[_i].arrInfo[E_Language.English].sName:="Line2Lift";
G_arrCylinder[_i].arrInfo[E_Language.Vietnamese].sName:="Xi lanh 2 lít đường ống";

_i:=E_Cylinder.Line2Prevent;
G_arrCylinder[_i].arrInfo[E_Language.Chinese].sName:="流水线2阻挡气缸";
G_arrCylinder[_i].arrInfo[E_Language.English].sName:="Line2Prevent";
G_arrCylinder[_i].arrInfo[E_Language.Vietnamese].sName:="Xi lanh chặn đường ống 2";

_i:=E_Cylinder.Line2Standard1;
G_arrCylinder[_i].arrInfo[E_Language.Chinese].sName:="流水线2校平气缸1";
G_arrCylinder[_i].arrInfo[E_Language.English].sName:="Line2Standard1";
G_arrCylinder[_i].arrInfo[E_Language.Vietnamese].sName:="Dòng 2 cân bằng xi lanh 1";

_i:=E_Cylinder.Line2Standard2;
G_arrCylinder[_i].arrInfo[E_Language.Chinese].sName:="流水线2校平气缸2";
G_arrCylinder[_i].arrInfo[E_Language.English].sName:="Line2Standard2";
G_arrCylinder[_i].arrInfo[E_Language.Vietnamese].sName:="Dòng 2 cân bằng xi lanh 2";

_i:=E_Cylinder.Line2OpenLateral1;
G_arrCylinder[_i].arrInfo[E_Language.Chinese].sName:="流水线2解锁侧推气缸1";
G_arrCylinder[_i].arrInfo[E_Language.English].sName:="Line2OpenLateral1";
G_arrCylinder[_i].arrInfo[E_Language.Vietnamese].sName:="Dòng 2 mở xi lanh đẩy bên 1";

_i:=E_Cylinder.Line2OpenRotate;
G_arrCylinder[_i].arrInfo[E_Language.Chinese].sName:="流水线2解锁旋转气缸";
G_arrCylinder[_i].arrInfo[E_Language.English].sName:="Line2OpenRotate";
G_arrCylinder[_i].arrInfo[E_Language.Vietnamese].sName:="Dây chuyền 2 mở khóa xi lanh xoay";

_i:=E_Cylinder.Line2OpenLateral2;
G_arrCylinder[_i].arrInfo[E_Language.Chinese].sName:="流水线2解锁侧推气缸2";
G_arrCylinder[_i].arrInfo[E_Language.English].sName:="Line2OpenLateral2";
G_arrCylinder[_i].arrInfo[E_Language.Vietnamese].sName:="Dây chuyền sản xuất 2 mở khóa xi lanh bên đẩy 2";

_i:=E_Cylinder.Line3LoadLift;
G_arrCylinder[_i].arrInfo[E_Language.Chinese].sName:="流水线3上料位顶升";
G_arrCylinder[_i].arrInfo[E_Language.English].sName:="Line3LoadLift";
G_arrCylinder[_i].arrInfo[E_Language.Vietnamese].sName:="Dòng 3 lên";

_i:=E_Cylinder.Line3LoadPrevent;
G_arrCylinder[_i].arrInfo[E_Language.Chinese].sName:="流水线3上料位阻挡";
G_arrCylinder[_i].arrInfo[E_Language.English].sName:="Line3LoadPrevent";
G_arrCylinder[_i].arrInfo[E_Language.Vietnamese].sName:="Dòng 3 lên cấp độ chặn";

_i:=E_Cylinder.Line3LoadRotate;
G_arrCylinder[_i].arrInfo[E_Language.Chinese].sName:="流水线3上料位旋转";
G_arrCylinder[_i].arrInfo[E_Language.English].sName:="Line3LoadRotate";
G_arrCylinder[_i].arrInfo[E_Language.Vietnamese].sName:="Dây chuyền sản xuất 3 cấp độ quay";

_i:=E_Cylinder.Line3OpenLift;
G_arrCylinder[_i].arrInfo[E_Language.Chinese].sName:="流水线3解锁位顶升";
G_arrCylinder[_i].arrInfo[E_Language.English].sName:="Line3OpenLift";
G_arrCylinder[_i].arrInfo[E_Language.Vietnamese].sName:="Dòng 3 mở khóa vị trí nâng lên";

_i:=E_Cylinder.Line3OpenPrevent;
G_arrCylinder[_i].arrInfo[E_Language.Chinese].sName:="流水线3解锁位阻挡";
G_arrCylinder[_i].arrInfo[E_Language.English].sName:="Line3OpenPrevent";
G_arrCylinder[_i].arrInfo[E_Language.Vietnamese].sName:="Dây chuyền 3 mở khóa vị trí chặn";

_i:=E_Cylinder.Line3Standard1;
G_arrCylinder[_i].arrInfo[E_Language.Chinese].sName:="流水线3校平气缸1";
G_arrCylinder[_i].arrInfo[E_Language.English].sName:="Line3Standard1";
G_arrCylinder[_i].arrInfo[E_Language.Vietnamese].sName:="Dòng 3 phẳng xi lanh 1";

_i:=E_Cylinder.Line3Standard2;
G_arrCylinder[_i].arrInfo[E_Language.Chinese].sName:="流水线3校平气缸2";
G_arrCylinder[_i].arrInfo[E_Language.English].sName:="Line3Standard2";
G_arrCylinder[_i].arrInfo[E_Language.Vietnamese].sName:="Dòng 3 cân bằng xi lanh 2";

_i:=E_Cylinder.Line3OpenLateral1;
G_arrCylinder[_i].arrInfo[E_Language.Chinese].sName:="流水线3解锁侧推气缸1";
G_arrCylinder[_i].arrInfo[E_Language.English].sName:="Line3OpenLateral1";
G_arrCylinder[_i].arrInfo[E_Language.Vietnamese].sName:="Dây chuyền sản xuất 3 mở khóa xi lanh bên đẩy 1";

_i:=E_Cylinder.Line3OpenRotate;
G_arrCylinder[_i].arrInfo[E_Language.Chinese].sName:="流水线3解锁旋转气缸";
G_arrCylinder[_i].arrInfo[E_Language.English].sName:="Line3OpenRotate";
G_arrCylinder[_i].arrInfo[E_Language.Vietnamese].sName:="Dây chuyền sản xuất 3 mở khóa xi lanh xoay";

_i:=E_Cylinder.Line3OpenLateral2;
G_arrCylinder[_i].arrInfo[E_Language.Chinese].sName:="流水线3解锁侧推气缸2";
G_arrCylinder[_i].arrInfo[E_Language.English].sName:="Line3OpenLateral2";
G_arrCylinder[_i].arrInfo[E_Language.Vietnamese].sName:="Dòng 3 mở khóa bên đẩy xi lanh 2";

_i:=E_Cylinder.TakeLift1;
G_arrCylinder[_i].arrInfo[E_Language.Chinese].sName:="取料模组升降气缸1";
G_arrCylinder[_i].arrInfo[E_Language.English].sName:="TakeLift1";
G_arrCylinder[_i].arrInfo[E_Language.Vietnamese].sName:="Lấy khối nâng xi lanh 1";

_i:=E_Cylinder.TakeLift2;
G_arrCylinder[_i].arrInfo[E_Language.Chinese].sName:="取料模组升降气缸2";
G_arrCylinder[_i].arrInfo[E_Language.English].sName:="TakeLift2";
G_arrCylinder[_i].arrInfo[E_Language.Vietnamese].sName:="Lấy khối nâng xi lanh 2";

_i:=E_Cylinder.TakeClamp;
G_arrCylinder[_i].arrInfo[E_Language.Chinese].sName:="取料模组夹紧气缸";
G_arrCylinder[_i].arrInfo[E_Language.English].sName:="TakeClamp";
G_arrCylinder[_i].arrInfo[E_Language.Vietnamese].sName:="Lấy mô-đun kẹp xi lanh";

_i:=E_Cylinder.UcLift;
G_arrCylinder[_i].arrInfo[E_Language.Chinese].sName:="下UC模组升降气缸";
G_arrCylinder[_i].arrInfo[E_Language.English].sName:="UcLift";
G_arrCylinder[_i].arrInfo[E_Language.Vietnamese].sName:="Xi lanh nâng theo mô-đun UC";

_i:=E_Cylinder.UcClamp;
G_arrCylinder[_i].arrInfo[E_Language.Chinese].sName:="下UC模组夹紧气缸";
G_arrCylinder[_i].arrInfo[E_Language.English].sName:="UcClamp";
G_arrCylinder[_i].arrInfo[E_Language.Vietnamese].sName:="Mô-đun dưới UC giữ chặt xi lanh";

_i:=E_Cylinder.UcSwing;
G_arrCylinder[_i].arrInfo[E_Language.Chinese].sName:="下UC模组摆动气缸";
G_arrCylinder[_i].arrInfo[E_Language.English].sName:="UcSwing";
G_arrCylinder[_i].arrInfo[E_Language.Vietnamese].sName:="Các xi lanh đang chuyển động trong mô-đun dưới UC";

_i:=E_Cylinder.UcLift1;
G_arrCylinder[_i].arrInfo[E_Language.Chinese].sName:="下UC升降气缸1";
G_arrCylinder[_i].arrInfo[E_Language.English].sName:="UcLift1";
G_arrCylinder[_i].arrInfo[E_Language.Vietnamese].sName:="Xi lanh nâng dưới UC 1";

_i:=E_Cylinder.UcClamp1;
G_arrCylinder[_i].arrInfo[E_Language.Chinese].sName:="下UC夹紧气缸1";
G_arrCylinder[_i].arrInfo[E_Language.English].sName:="UcClamp1";
G_arrCylinder[_i].arrInfo[E_Language.Vietnamese].sName:="Dưới ống 1";

_i:=E_Cylinder.UcRotate1;
G_arrCylinder[_i].arrInfo[E_Language.Chinese].sName:="下UC旋转气缸1";
G_arrCylinder[_i].arrInfo[E_Language.English].sName:="UcRotate1";
G_arrCylinder[_i].arrInfo[E_Language.Vietnamese].sName:="Xi lanh xoay phía dưới UC 1";

_i:=E_Cylinder.UcLift2;
G_arrCylinder[_i].arrInfo[E_Language.Chinese].sName:="下UC升降气缸2";
G_arrCylinder[_i].arrInfo[E_Language.English].sName:="UcLift2";
G_arrCylinder[_i].arrInfo[E_Language.Vietnamese].sName:="Nâng xi lanh 2";

_i:=E_Cylinder.UcClamp2;
G_arrCylinder[_i].arrInfo[E_Language.Chinese].sName:="下UC夹紧气缸2";
G_arrCylinder[_i].arrInfo[E_Language.English].sName:="UcClamp2";
G_arrCylinder[_i].arrInfo[E_Language.Vietnamese].sName:="Dưới ống 2";

_i:=E_Cylinder.UcRotate2;
G_arrCylinder[_i].arrInfo[E_Language.Chinese].sName:="下UC旋转气缸2";
G_arrCylinder[_i].arrInfo[E_Language.English].sName:="UcRotate2";
G_arrCylinder[_i].arrInfo[E_Language.Vietnamese].sName:="Xi lanh quay dưới UC 2";

_i:=E_Cylinder.UcDrive;
G_arrCylinder[_i].arrInfo[E_Language.Chinese].sName:="下UC皮带推料气缸";
G_arrCylinder[_i].arrInfo[E_Language.English].sName:="UcDrive";
G_arrCylinder[_i].arrInfo[E_Language.Vietnamese].sName:="Ống đẩy dưới vành đai UC";

_i:=E_Cylinder.FrockElevator1;
G_arrCylinder[_i].arrInfo[E_Language.Chinese].sName:="下工装提升气缸1";
G_arrCylinder[_i].arrInfo[E_Language.English].sName:="FrockElevator1";
G_arrCylinder[_i].arrInfo[E_Language.Vietnamese].sName:="Máy nâng xi lanh 1";

_i:=E_Cylinder.FrockRotateDown1;
G_arrCylinder[_i].arrInfo[E_Language.Chinese].sName:="下工装旋转压紧气缸1";
G_arrCylinder[_i].arrInfo[E_Language.English].sName:="FrockRotateDown1";
G_arrCylinder[_i].arrInfo[E_Language.Vietnamese].sName:="Tải trọng xoay xi lanh 1";

_i:=E_Cylinder.FrockPush1;
G_arrCylinder[_i].arrInfo[E_Language.Chinese].sName:="下工装拨料气缸1";
G_arrCylinder[_i].arrInfo[E_Language.English].sName:="FrockPush1";
G_arrCylinder[_i].arrInfo[E_Language.Vietnamese].sName:="Xi lanh máy đo 1";

_i:=E_Cylinder.FrockElevator2;
G_arrCylinder[_i].arrInfo[E_Language.Chinese].sName:="下工装提升气缸2";
G_arrCylinder[_i].arrInfo[E_Language.English].sName:="FrockElevator2";
G_arrCylinder[_i].arrInfo[E_Language.Vietnamese].sName:="";

_i:=E_Cylinder.FrockRotateDown2;
G_arrCylinder[_i].arrInfo[E_Language.Chinese].sName:="下工装旋转压紧气缸2";
G_arrCylinder[_i].arrInfo[E_Language.English].sName:="FrockRotateDown2";
G_arrCylinder[_i].arrInfo[E_Language.Vietnamese].sName:="";

_i:=E_Cylinder.FrockPush2;
G_arrCylinder[_i].arrInfo[E_Language.Chinese].sName:="下工装拨料气缸2";
G_arrCylinder[_i].arrInfo[E_Language.English].sName:="FrockPush2";
G_arrCylinder[_i].arrInfo[E_Language.Vietnamese].sName:="";

_i:=E_Cylinder.FrockBelt;
G_arrCylinder[_i].arrInfo[E_Language.Chinese].sName:="下工装皮带推料气缸";
G_arrCylinder[_i].arrInfo[E_Language.English].sName:="FrockBelt";
G_arrCylinder[_i].arrInfo[E_Language.Vietnamese].sName:="";
END_ACTION

ACTION A_InOut:
FOR _i:=0 TO 7 BY 1 DO
	FOR _t:=0 TO 15 BY 1 DO
		IF GVL.stSetting.bDryRun AND ((_i=6 AND _t>=6) OR _i>6) THEN
			_fbPulse(PT:=T#1S , Q=> _arrInput[_i,_t]);
		ELSE
			_arrTonInput[_i,_t](IN:=GVL_IO.I[_i,_t] , PT:=TO_TIME(GVL_Data.stRecipe.arrInputTon[_i,_t]) , Q=>_arrInput[_i,_t] , ET=> );
		END_IF
	END_FOR
END_FOR

FOR _i:=0 TO 6 BY 1 DO
	FOR _t:=0 TO 15 BY 1 DO
		IF NOT G_stSystem.stMode.bSetting THEN
			_arrTonOutput[_i,_t](IN:=_arrOutput[_i,_t] , PT:=TO_TIME(GVL_Data.stRecipe.arrOutputTon[_i,_t]) , Q=>GVL_IO.Q[_i,_t] , ET=> );
		END_IF
	END_FOR
END_FOR

Data_TO_Data(ADR(_arrInput),SIZEOF(_arrInput),ADR(GVL.I),SIZEOF(GVL.I));
Data_TO_Data(ADR(GVL.Q),SIZEOF(GVL.Q),ADR(_arrOutput),SIZEOF(_arrOutput));



CASE GVL_Data.stRecipe.eMachineType OF
	E_MachineType.LH311,E_MachineType.RH311:
		FOR _i:=3 TO 4 BY 1 DO
			GVL.stShield_Q[2,_i]:=GVL.stShield_I[2,_i]:=TRUE;
		END_FOR
		FOR _i:=9 TO 10 BY 1 DO
			GVL.stShield_Q[3,_i]:=GVL.stShield_I[3,_i]:=TRUE;
		END_FOR
		FOR _i:=9 TO 15 BY 1 DO
			GVL.stShield_Q[4,_i]:=GVL.stShield_I[4,_i]:=TRUE;
		END_FOR
		FOR _i:=0 TO 6 BY 1 DO
			GVL.stShield_Q[5,_i]:=GVL.stShield_I[5,_i]:=TRUE;
		END_FOR
		GVL.stShield_Q[6,9]:=TRUE;
		FOR _i:=6 TO 9 BY 1 DO
			GVL.stShield_I[7,_i]:=TRUE;
		END_FOR
	E_MachineType.LH353,E_MachineType.RH353:
		FOR _i:=13 TO 14 BY 1 DO
			GVL.stShield_Q[1,_i]:=GVL.stShield_I[1,_i]:=TRUE;
		END_FOR
		FOR _i:=3 TO 4 BY 1 DO
			GVL.stShield_Q[3,_i]:=GVL.stShield_I[3,_i]:=TRUE;
		END_FOR
		FOR _i:=13 TO 15 BY 1 DO
			GVL.stShield_Q[3,_i]:=GVL.stShield_I[3,_i]:=TRUE;
		END_FOR
		GVL.stShield_Q[4,0]:=GVL.stShield_I[4,0]:=TRUE;
		FOR _i:=3 TO 8 BY 1 DO
			GVL.stShield_Q[4,_i]:=GVL.stShield_I[4,_i]:=TRUE;
		END_FOR
		GVL.stShield_I[7,5]:=TRUE;
	E_MachineType.LH367,E_MachineType.RH367:
		FOR _i:=13 TO 14 BY 1 DO
			GVL.stShield_Q[1,_i]:=GVL.stShield_I[1,_i]:=TRUE;
		END_FOR
		FOR _i:=3 TO 4 BY 1 DO
			GVL.stShield_Q[3,_i]:=GVL.stShield_I[3,_i]:=TRUE;
		END_FOR
		FOR _i:=3 TO 8 BY 1 DO
			GVL.stShield_Q[4,_i]:=GVL.stShield_I[4,_i]:=TRUE;
		END_FOR
		GVL.stShield_I[7,5]:=TRUE;
	E_MachineType.LH201,E_MachineType.RH201:
		FOR _i:=11 TO 14 BY 1 DO
			GVL.stShield_Q[1,_i]:=GVL.stShield_I[1,_i]:=TRUE;
		END_FOR
		FOR _i:=1 TO 4 BY 1 DO
			GVL.stShield_Q[3,_i]:=GVL.stShield_I[3,_i]:=TRUE;
		END_FOR
		FOR _i:=13 TO 15 BY 1 DO
			GVL.stShield_Q[3,_i]:=GVL.stShield_I[3,_i]:=TRUE;
		END_FOR
		GVL.stShield_Q[4,0]:=GVL.stShield_I[4,0]:=TRUE;
		FOR _i:=3 TO 8 BY 1 DO
			GVL.stShield_Q[4,_i]:=GVL.stShield_I[4,_i]:=TRUE;
		END_FOR
		GVL.stShield_I[7,5]:=TRUE;
	E_MachineType.LH069,E_MachineType.RH069:
		FOR _i:=11 TO 14 BY 1 DO
			GVL.stShield_Q[1,_i]:=GVL.stShield_I[1,_i]:=TRUE;
		END_FOR
		FOR _i:=1 TO 4 BY 1 DO
			GVL.stShield_Q[3,_i]:=GVL.stShield_I[3,_i]:=TRUE;
		END_FOR
		FOR _i:=13 TO 15 BY 1 DO
			GVL.stShield_Q[3,_i]:=GVL.stShield_I[3,_i]:=TRUE;
		END_FOR
		GVL.stShield_Q[4,0]:=GVL.stShield_I[4,0]:=TRUE;
		FOR _i:=3 TO 8 BY 1 DO
			GVL.stShield_Q[4,_i]:=GVL.stShield_I[4,_i]:=TRUE;
		END_FOR
		GVL.stShield_I[7,5]:=TRUE;
	E_MachineType.LH373,E_MachineType.RH373:
		FOR _i:=13 TO 14 BY 1 DO
			GVL.stShield_Q[1,_i]:=GVL.stShield_I[1,_i]:=TRUE;
		END_FOR
		FOR _i:=3 TO 4 BY 1 DO
			GVL.stShield_Q[2,_i]:=GVL.stShield_I[2,_i]:=TRUE;
		END_FOR
		FOR _i:=3 TO 4 BY 1 DO
			GVL.stShield_Q[3,_i]:=GVL.stShield_I[3,_i]:=TRUE;
		END_FOR
		FOR _i:=13 TO 15 BY 1 DO
			GVL.stShield_Q[3,_i]:=GVL.stShield_I[3,_i]:=TRUE;
		END_FOR
		GVL.stShield_Q[4,0]:=GVL.stShield_I[4,0]:=TRUE;
		FOR _i:=3 TO 8 BY 1 DO
			GVL.stShield_Q[4,_i]:=GVL.stShield_I[4,_i]:=TRUE;
		END_FOR
		GVL.stShield_I[7,5]:=TRUE;
END_CASE
END_ACTION

ACTION A_Line:
GVL.arrFbLine[E_Line.Line1](System:=G_stSystem , Moving=>GVL.Q.bLine1Axis );

GVL.arrFbLine[E_Line.Line2](System:=G_stSystem , Moving=>GVL.Q.bLine2Axis  );

GVL.arrFbLine[E_Line.Line3](System:=G_stSystem , Moving=>GVL.Q.bLine3Axis );

GVL.arrFbLine[E_Line.UnloadElevator](System:=G_stSystem , Moving=>GVL.Q.bUnloadElevatorLine );

GVL.arrFbLine[E_Line.UnloadUC](System:=G_stSystem , Moving=>GVL.Q.bUnloadUCLine );


_homeLineTon(IN:=G_stSystem.stMode.bHoming, PT:=GVL.stSetting.tHomeLine , Q=> , ET=> );

IF G_stSystem.stMode.bAutoRunning THEN
	GVL.arrFbLine[E_Line.Line1].M_Jog(1);
	GVL.arrFbLine[E_Line.Line2].M_Jog(1);
	GVL.arrFbLine[E_Line.Line3].M_Jog(1);
END_IF
END_ACTION

END_PROGRAM

// ---- POUs/P_Station.TcPOU
PROGRAM P_Station
VAR
	_stParameter:				ST_StationParameter;
	_stHandshake:				ST_StationHandshake;
	
	_fbTakeLoad:				FB_StationTakeLoad;// 取料站
	_fbDismantling_L2:			FB_StationDismantling;// 线体2 拆解站 
	_fbDismantling_L3:			FB_StationDismantling;// 线体3 拆解站 
	_fbLine0Load:				FB_StationLine0Load;// 线体0 上料站
	_fbLine0Buffer:				FB_StationLine0Buffer;// 线体0 缓存站
	_fbLineLoad_L1:				FB_StationLineLoad;// 线体1 上料站
	_fbLineLoad_L3:				FB_StationLineLoad;// 线体3 上料站
	_fbUnloadUc_L2:				FB_StationUnloadUc;// 线体2 下UC
	_fbUnloadUc_L3:				FB_StationUnloadUc;// 线体3 下UC
	_fbUnloadElevator_L2:		FB_StationUnloadElevator;// 线体2 下工装
	_fbUnloadElevator_L3:		FB_StationUnloadElevator;// 线体3 下工装
	_fbUnloadLineUc:			FB_StationUnloadLine;//下UC 线体
	_fbUnloadLineElevator:		FB_StationUnloadLine;// 下工装线体
	_fbStationUnLoadUc_311:		FB_StationUnLoadUc_311;// 下UC 模组
		
	_vArrFbCylinder:			ARRAY[0..10] OF FB_Cylinder;// 虚拟气缸
	_vArrCylinder:				ARRAY[0..10] OF ST_Cylinder;// 虚拟气缸
	_vArrCylinderData:			ARRAY[0..10] OF ST_CylinderData;// 虚拟气缸
	_i:							INT;
	_bFistRun:					BOOL:=true;
END_VAR

GVL.stSetting.eTakeMode:=M_LoadPriority(_stParameter,GVL_Data.stRecipe);
IF _bFistRun THEN
	A_Info();
	_bFistRun:=FALSE;
END_IF


A_Handshake();// 交握

A_Virtual();// 虚拟硬件



A_TakeLoad();// 取料站

A_Dismantling_L2();// 拆解站

A_Dismantling_L3();// 拆解站

A_Line0Buffer();// 线体0 上料缓存

A_Line0Load();// 线体0 上料站

A_LineLoad_L1();// 线体1 上料

A_LineLoad_L3();// 线体3 上料

A_UnloadElevator_L2();// 线体2 下工装

A_UnloadElevator_L3();// 线体3 下工装

A_UnloadLineElevator();// 下工装 流线

A_UnLoadUc_311();// 下UC模组  紧311使用

A_UnloadLineUc();// 下UC 流线 311以为下料程序

A_UnloadUc_L2();// 线体2下UC 311以外下料程序

A_UnloadUc_L3();// 线体3 下UC 311以为下料程序

ACTION A_Dismantling_L2:
_stParameter.stLine2Dismantling.bPalletCheck1:=GVL.I.bLine2PalletCheck1;
_stParameter.stLine2Dismantling.bPalletCheck2:=GVL.I.bLine2PalletCheck2;
_stParameter.stLine2Dismantling.bPalletCheck3:=GVL.I.bLine2PalletCheck3;
_stParameter.stLine2Dismantling.fbLateral1 REF=G_arrFbCylinder[E_Cylinder.Line2OpenLateral1];
_stParameter.stLine2Dismantling.fbLateral2 REF=G_arrFbCylinder[E_Cylinder.Line2OpenLateral2];
_stParameter.stLine2Dismantling.fbLift REF= G_arrFbCylinder[E_Cylinder.Line2Lift];
_stParameter.stLine2Dismantling.fbPrevent REF= G_arrFbCylinder[E_Cylinder.Line2Prevent];
_stParameter.stLine2Dismantling.fbRotate REF= G_arrFbCylinder[E_Cylinder.Line2OpenRotate];
_stParameter.stLine2Dismantling.fbStandard1 REF= G_arrFbCylinder[E_Cylinder.Line2Standard1];
_stParameter.stLine2Dismantling.fbStandard2 REF= G_arrFbCylinder[E_Cylinder.Line2Standard2];
_stParameter.stLine2Dismantling.bClose:=GVL_Data.stRecipe.eLineClose=E_LineClose.Line2;
_stParameter.stLine2Dismantling.bCloseUnloadElevator:=FALSE;

_fbDismantling_L2(
	Enable:=TRUE,
	System:=G_stSystem , 
	Station:=G_arrStation[E_Station.Line2Dismantling] , 
	Error:=G_stError , 
	Setting:=GVL.stSetting , 
	Recipe:=GVL_Data.stRecipe , 
	Parameter:=_stParameter.stLine2Dismantling);
END_ACTION

ACTION A_Dismantling_L3:
_stParameter.stLine3Dismantling.bPalletCheck1:=GVL.I.bLine3OpenCheck1;
_stParameter.stLine3Dismantling.bPalletCheck2:=GVL.I.bLine3OpenCheck2;
_stParameter.stLine3Dismantling.bPalletCheck3:=GVL.I.bLine3OpenCheck3;
_stParameter.stLine3Dismantling.fbLateral1 REF=G_arrFbCylinder[E_Cylinder.Line3OpenLateral1];
_stParameter.stLine3Dismantling.fbLateral2 REF=G_arrFbCylinder[E_Cylinder.Line3OpenLateral2];
_stParameter.stLine3Dismantling.fbLift REF= G_arrFbCylinder[E_Cylinder.Line3OpenLift];
_stParameter.stLine3Dismantling.fbPrevent REF= G_arrFbCylinder[E_Cylinder.Line3OpenPrevent];
_stParameter.stLine3Dismantling.fbRotate REF= G_arrFbCylinder[E_Cylinder.Line3OpenRotate];
_stParameter.stLine3Dismantling.fbStandard1 REF= G_arrFbCylinder[E_Cylinder.Line3Standard1];
_stParameter.stLine3Dismantling.fbStandard2 REF= G_arrFbCylinder[E_Cylinder.Line3Standard2];
_stParameter.stLine3Dismantling.bClose:=GVL_Data.stRecipe.eLineClose=E_LineClose.Line3;
_stParameter.stLine3Dismantling.bCloseUnloadElevator:=FALSE;

_fbDismantling_L3(
	Enable:=TRUE,
	System:=G_stSystem , 
	Station:=G_arrStation[E_Station.Line3Dismantling] , 
	Error:=G_stError , 
	Setting:=GVL.stSetting , 
	Recipe:=GVL_Data.stRecipe , 
	Parameter:=_stParameter.stLine3Dismantling);
END_ACTION

ACTION A_Handshake:
_stParameter.stLine0Load.stHandshake.bRequestLine0Load:=_stParameter.stLine0Buffer.stHandshake.bRequestLine0Load;

_stParameter.stLine0Buffer.stHandshake.bRequestLine0Buffer_T:=_stParameter.stTakeLoad.stHandshake.bRequestLine0Buffer_T0;
_stParameter.stLine0Buffer.stHandshake.bResponseLine0Buffer:=_stParameter.stLine0Load.stHandshake.bResponseLine0Buffer;

_stParameter.stLine1Load.stHandshake.bRequestLineLoad_D:=_stParameter.stLine2Dismantling.stHandshake.bRequestLineLoad_D;
_stParameter.stLine1Load.stHandshake.bRequestLineLoad_P:=_stParameter.stTakeLoad.stHandshake.bRequestLineLoad_P1;
_stParameter.stLine1Load.stHandshake.bRequestLineLoad_T:=_stParameter.stTakeLoad.stHandshake.bRequestLineLoad_T1;
_stParameter.stLine1Load.stHandshake.bRequestTake_P_M:=FALSE;
_stParameter.stLine1Load.stHandshake.bResponseMachine_P:=FALSE;

_stParameter.stLine2UnloadElevator.stHandshake.bRequestElevator:=_stParameter.stLine2Dismantling.stHandshake.bRequestElevator;
_stParameter.stLine2UnloadElevator.stHandshake.bResponseElevator:=_stParameter.stUnloadLineElevator.stHandshake.bResponseUnladLine2;

_stParameter.stLine2UnloadUc.stHandshake.bResponseUnladLine:=_stParameter.stUnloadLineUc.stHandshake.bResponseUnladLine2;

_stParameter.stLine3Load.stHandshake.bRequestLineLoad_D:=_stParameter.stLine3Dismantling.stHandshake.bRequestLineLoad_D;
_stParameter.stLine3Load.stHandshake.bRequestLineLoad_P:=_stParameter.stTakeLoad.stHandshake.bRequestLineLoad_P3;
_stParameter.stLine3Load.stHandshake.bRequestLineLoad_T:=_stParameter.stTakeLoad.stHandshake.bRequestLineLoad_T3;
_stParameter.stLine3Load.stHandshake.bRequestTake_P_M:=FALSE;
_stParameter.stLine3Load.stHandshake.bResponseMachine_P:=FALSE;

_stParameter.stLine3UnloadElevator.stHandshake.bRequestElevator:=_stParameter.stLine3Dismantling.stHandshake.bRequestElevator;
_stParameter.stLine3UnloadElevator.stHandshake.bResponseElevator:=_stParameter.stUnloadLineElevator.stHandshake.bResponseUnladLine3;

_stParameter.stLine3UnloadUc.stHandshake.bResponseUnladLine:=_stParameter.stUnloadLineUc.stHandshake.bResponseUnladLine3;

_stParameter.stTakeLoad.stHandshake.bResponseTake_P1:=_stParameter.stLine1Load.stHandshake.bResponseTake_P;
_stParameter.stTakeLoad.stHandshake.bResponseTake_P3:=_stParameter.stLine3Load.stHandshake.bResponseTake_P;
_stParameter.stTakeLoad.stHandshake.bResponseTake_T0:=_stParameter.stLine0Buffer.stHandshake.bResponseTake_T;
_stParameter.stTakeLoad.stHandshake.bResponseTake_T1:=_stParameter.stLine1Load.stHandshake.bResponseTake_T;
_stParameter.stTakeLoad.stHandshake.bResponseTake_T3:=_stParameter.stLine3Load.stHandshake.bResponseTake_T;

_stParameter.stUnloadLineElevator.stHandshake.bRequestUnloadLine2:=_stParameter.stLine2UnloadElevator.stHandshake.bRequestUnline;
_stParameter.stUnloadLineElevator.stHandshake.bRequestUnloadLine3:=_stParameter.stLine3UnloadElevator.stHandshake.bRequestUnline;

_stParameter.stUnloadLineUc.stHandshake.bRequestUnloadLine2:=_stParameter.stLine2UnloadUc.stHandshake.bRequestUnloadLine;
_stParameter.stUnloadLineUc.stHandshake.bRequestUnloadLine3:=_stParameter.stLine3UnloadUc.stHandshake.bRequestUnloadLine;

_stParameter.stLine2Dismantling.stHandshake.bResponseDismantling_D:=_stParameter.stLine1Load.stHandshake.bResponseDismantling_D;
_stParameter.stLine2Dismantling.stHandshake.bResponseDismantling_E:=_stParameter.stLine2UnloadElevator.stHandshake.bResponseDismantling_E;
_stParameter.stLine3Dismantling.stHandshake.bResponseDismantling_D:=_stParameter.stLine3Load.stHandshake.bResponseDismantling_D;
_stParameter.stLine3Dismantling.stHandshake.bResponseDismantling_E:=_stParameter.stLine3UnloadElevator.stHandshake.bResponseDismantling_E;

IF GVL_Data.stRecipe.eMachineType =E_MachineType.RH311 OR GVL_Data.stRecipe.eMachineType =E_MachineType.LH311 THEN
	_stParameter.stUnloadUc_311.stHandshake.bRequestUc_L2:=_stParameter.stLine2Dismantling.stHandshake.bRequestUc;
	_stParameter.stUnloadUc_311.stHandshake.bRequestUc_L3:=_stParameter.stLine3Dismantling.stHandshake.bRequestUc;
	_stParameter.stLine2Dismantling.stHandshake.bResponseDismantling_Uc:=_stParameter.stUnloadUc_311.stHandshake.bResponseDismantling_Uc_L2;
	_stParameter.stLine3Dismantling.stHandshake.bResponseDismantling_Uc:=_stParameter.stUnloadUc_311.stHandshake.bResponseDismantling_Uc_L3;
ELSE
	_stParameter.stLine2UnloadUc.stHandshake.bRequestUc:=_stParameter.stLine2Dismantling.stHandshake.bRequestUc;
	_stParameter.stLine3UnloadUc.stHandshake.bRequestUc:=_stParameter.stLine3Dismantling.stHandshake.bRequestUc;
	_stParameter.stLine2Dismantling.stHandshake.bResponseDismantling_Uc:=_stParameter.stLine2UnloadUc.stHandshake.bResponseDismantling_Uc;
	_stParameter.stLine3Dismantling.stHandshake.bResponseDismantling_Uc:=_stParameter.stLine3UnloadUc.stHandshake.bResponseDismantling_Uc;
END_IF
END_ACTION

ACTION A_Info:
_i:=E_Station.Line0Load;
G_arrStation[_i].arrName[E_Language.Chinese]:="主流线上料工站";
G_arrStation[_i].arrName[E_Language.English]:="Line0Load";
G_arrStation[_i].arrName[E_Language.Vietnamese]:="Trạm vật liệu dòng chính";

_i:=E_Station.Line0Buffer;
G_arrStation[_i].arrName[E_Language.Chinese]:="主流线缓存工站";
G_arrStation[_i].arrName[E_Language.English]:="Line0Buffer";
G_arrStation[_i].arrName[E_Language.Vietnamese]:="Trạm bộ nhớ nhớ đường chính";

_i:=E_Station.TakeLoad;
G_arrStation[_i].arrName[E_Language.Chinese]:="上料取料工站";
G_arrStation[_i].arrName[E_Language.English]:="TakeLoad";
G_arrStation[_i].arrName[E_Language.Vietnamese]:="Nhà ga ăn uống";

_i:=E_Station.Line3Load;
G_arrStation[_i].arrName[E_Language.Chinese]:="流线3上料工站";
G_arrStation[_i].arrName[E_Language.English]:="Line3Load";
G_arrStation[_i].arrName[E_Language.Vietnamese]:="Trạm sạc 3 dòng";

_i:=E_Station.Line1Load;
G_arrStation[_i].arrName[E_Language.Chinese]:="流线2上料工站";
G_arrStation[_i].arrName[E_Language.English]:="Line1Load";
G_arrStation[_i].arrName[E_Language.Vietnamese]:="Trạm lên men dòng 2";

_i:=E_Station.Line2Dismantling;
G_arrStation[_i].arrName[E_Language.Chinese]:="流线2拆解工站";
G_arrStation[_i].arrName[E_Language.English]:="Line2Dismantling";
G_arrStation[_i].arrName[E_Language.Vietnamese]:="Trạm tháo dỡ dòng 2";

_i:=E_Station.Line3Dismantling;
G_arrStation[_i].arrName[E_Language.Chinese]:="流线3拆解工站";
G_arrStation[_i].arrName[E_Language.English]:="Line3Dismantling";
G_arrStation[_i].arrName[E_Language.Vietnamese]:="Trạm tháo dỡ dòng 3";

_i:=E_Station.Line2UnloadElevator;
G_arrStation[_i].arrName[E_Language.Chinese]:="线体2下工装";
G_arrStation[_i].arrName[E_Language.English]:="Line2UnloadElevator";
G_arrStation[_i].arrName[E_Language.Vietnamese]:="Thiết bị dây chuyền 2";

_i:=E_Station.Line3UnloadElevator;
G_arrStation[_i].arrName[E_Language.Chinese]:="线体3下工装";
G_arrStation[_i].arrName[E_Language.English]:="Line3UnloadElevator";
G_arrStation[_i].arrName[E_Language.Vietnamese]:="Dây số 3 dưới công cụ";

_i:=E_Station.Line2UnloadUc;
G_arrStation[_i].arrName[E_Language.Chinese]:="线体2 下UC";
G_arrStation[_i].arrName[E_Language.English]:="Line2UnloadUc";
G_arrStation[_i].arrName[E_Language.Vietnamese]:="Máy dò 2 ở UC";

_i:=E_Station.Line3UnloadUc;
G_arrStation[_i].arrName[E_Language.Chinese]:="线体3 下UC";
G_arrStation[_i].arrName[E_Language.English]:="Line3UnloadUc";
G_arrStation[_i].arrName[E_Language.Vietnamese]:="Máy dò 3 ở UC";

_i:=E_Station.UnloadLineUc;
G_arrStation[_i].arrName[E_Language.Chinese]:="下UC 线体";
G_arrStation[_i].arrName[E_Language.English]:="UnloadLineUc";
G_arrStation[_i].arrName[E_Language.Vietnamese]:="Ống dẫn dưới UC";

_i:=E_Station.UnloadLineElevator;
G_arrStation[_i].arrName[E_Language.Chinese]:="下工装 线体";
G_arrStation[_i].arrName[E_Language.English]:="UnloadLineElevator";
G_arrStation[_i].arrName[E_Language.Vietnamese]:="Thiết bị dây";

_i:=E_Station.UnloadUc_311;
G_arrStation[_i].arrName[E_Language.Chinese]:="下UC模组";
G_arrStation[_i].arrName[E_Language.English]:="UnloadUc_311";
G_arrStation[_i].arrName[E_Language.Vietnamese]:="Mô-đun dưới UC";
END_ACTION

ACTION A_Line0Buffer:

_stParameter.stLine0Buffer.bPlace:=GVL.I.bLine0Place;


_fbLine0Buffer(
	Enable:=TRUE,
	System:=G_stSystem , 
	Station:=G_arrStation[E_Station.Line0Buffer] , 
	Error:=G_stError , 
	Setting:=GVL.stSetting , 
	Recipe:=GVL_Data.stRecipe , 
	Parameter:=_stParameter.stLine0Buffer);
END_ACTION

ACTION A_Line0Load:
_stParameter.stLine0Load.bPartCheck:=GVL.I.bLine0Part;
_stParameter.stLine0Load.bPreventCheck:=GVL.I.bLine0Prevent;
_stParameter.stLine0Load.fbPart REF= G_arrFbCylinder[E_Cylinder.Line0Part];
_stParameter.stLine0Load.fbPrevent REF= G_arrFbCylinder[E_Cylinder.Line0Prevent];

_fbLine0Load(
	Enable:=TRUE,
	System:=G_stSystem , 
	Station:=G_arrStation[E_Station.Line0Load] , 
	Error:=G_stError , 
	Setting:=GVL.stSetting , 
	Recipe:=GVL_Data.stRecipe , 
	Parameter:=_stParameter.stLine0Load);
END_ACTION

ACTION A_LineLoad_L1:
_stParameter.stLine1Load.bIsClosed:=GVL_Data.stRecipe.eLoadClose=E_LoadClose.Line1;
_stParameter.stLine1Load.bIsPlacing:=GVL.stSetting.eTakeModeBuffer=E_TakeMode.Place1;
_stParameter.stLine1Load.bIsTaking:=GVL.stSetting.eTakeModeBuffer=E_TakeMode.Take1;
_stParameter.stLine1Load.bPalletCheck1:=GVL.I.bLine1PalletCheck1;
_stParameter.stLine1Load.bPalletCheck2:=GVL.I.bLine1PalletCheck2;
_stParameter.stLine1Load.bPalletCheck3:=GVL.I.bLine1PalletCheck3;
_stParameter.stLine1Load.fbAdjust1 REF= G_arrFbCylinder[E_Cylinder.Line1Adjust1];
_stParameter.stLine1Load.fbElevator REF= G_arrFbCylinder[E_Cylinder.Line1Elevator];
_stParameter.stLine1Load.fbLift REF= G_arrFbCylinder[E_Cylinder.Line1Lift];
_stParameter.stLine1Load.fbPrevent REF= G_arrFbCylinder[E_Cylinder.Line1Prevent];
_stParameter.stLine1Load.fbRotate REF= G_arrFbCylinder[E_Cylinder.Line1Rotate];
_stParameter.stLine1Load.bManualLoad:=FALSE;
_fbLineLoad_L1(
	Enable:=true,
	System:=G_stSystem , 
	Station:=G_arrStation[E_Station.Line1Load] , 
	Error:=G_stError , 
	Setting:=GVL.stSetting , 
	Recipe:=GVL_Data.stRecipe , 
	Parameter:=_stParameter.stLine1Load);
END_ACTION

ACTION A_LineLoad_L3:
_stParameter.stLine3Load.bIsClosed:=FALSE;
_stParameter.stLine3Load.bIsPlacing:=GVL.stSetting.eTakeModeBuffer=E_TakeMode.Place3Load;
_stParameter.stLine3Load.bIsTaking:=GVL.stSetting.eTakeModeBuffer=E_TakeMode.Take3Load;
_stParameter.stLine3Load.bPalletCheck1:=GVL.I.bLine3PalletCheck1;
_stParameter.stLine3Load.bPalletCheck2:=GVL.I.bLine3PalletCheck2;
_stParameter.stLine3Load.bPalletCheck3:=GVL.I.bLine3PalletCheck3;
_stParameter.stLine3Load.fbAdjust1 REF= _vArrFbCylinder[0];
_stParameter.stLine3Load.fbElevator REF=_vArrFbCylinder[1];
_stParameter.stLine3Load.fbLift REF= G_arrFbCylinder[E_Cylinder.Line3LoadLift];
_stParameter.stLine3Load.fbPrevent REF= G_arrFbCylinder[E_Cylinder.Line3LoadPrevent];
_stParameter.stLine3Load.fbRotate REF= G_arrFbCylinder[E_Cylinder.Line3LoadRotate];
_stParameter.stLine3Load.bManualLoad:=FALSE;

_fbLineLoad_L3(
	Enable:=TRUE,
	System:=G_stSystem , 
	Station:=G_arrStation[E_Station.Line3Load] , 
	Error:=G_stError , 
	Setting:=GVL.stSetting , 
	Recipe:=GVL_Data.stRecipe , 
	Parameter:=_stParameter.stLine3Load);
END_ACTION

ACTION A_TakeLoad:
_stParameter.stTakeLoad.fbTakeClamp REF= G_arrFbCylinder[E_Cylinder.TakeClamp];
_stParameter.stTakeLoad.fbTakeLift1 REF= G_arrFbCylinder[E_Cylinder.TakeLift1];
_stParameter.stTakeLoad.fbTakeLift2 REF= G_arrFbCylinder[E_Cylinder.TakeLift2];
_stParameter.stTakeLoad.fbTakeY REF= G_arrFbAxis[E_Axis.TakeY];
_stParameter.stTakeLoad.fbTakeZ REF= G_arrFbAxis[E_Axis.TakeZ];

_fbTakeLoad(
	Enable:=TRUE,
	System:=G_stSystem , 
	Station:=G_arrStation[E_Station.TakeLoad] , 
	Error:=G_stError , 
	Setting:=GVL.stSetting , 
	Recipe:=GVL_Data.stRecipe , 
	Parameter:=_stParameter.stTakeLoad);
END_ACTION

ACTION A_UnloadElevator_L2:
_stParameter.stLine2UnloadElevator.bFrockElevator1NoneCheck:=GVL.I.bFrockElevator1NoneCheck;
_stParameter.stLine2UnloadElevator.fbFrockElevator REF= G_arrFbCylinder[E_Cylinder.FrockElevator1];
_stParameter.stLine2UnloadElevator.fbFrockPush REF= G_arrFbCylinder[E_Cylinder.FrockPush1];
_stParameter.stLine2UnloadElevator.fbFrockRotateDown REF= G_arrFbCylinder[E_Cylinder.FrockRotateDown1];
_stParameter.stLine2UnloadElevator.bManualUnload:=FALSE;


_fbUnloadElevator_L2(
	Enable:=TRUE,
	System:=G_stSystem , 
	Station:=G_arrStation[E_Station.Line2UnloadElevator] , 
	Error:=G_stError , 
	Setting:=GVL.stSetting , 
	Recipe:=GVL_Data.stRecipe , 
	Parameter:=_stParameter.stLine2UnloadElevator);
END_ACTION

ACTION A_UnloadElevator_L3:

_stParameter.stLine3UnloadElevator.bFrockElevator1NoneCheck:=GVL.I.bFrockElevator2NoneCheck;
_stParameter.stLine3UnloadElevator.fbFrockElevator REF= G_arrFbCylinder[E_Cylinder.FrockElevator2];
_stParameter.stLine3UnloadElevator.fbFrockPush REF= G_arrFbCylinder[E_Cylinder.FrockPush2];
_stParameter.stLine3UnloadElevator.fbFrockRotateDown REF= G_arrFbCylinder[E_Cylinder.FrockRotateDown2];
_stParameter.stLine3UnloadElevator.bManualUnload:=FALSE;

_fbUnloadElevator_L3(
	Enable:=TRUE,
	System:=G_stSystem , 
	Station:=G_arrStation[E_Station.Line3UnloadElevator] , 
	Error:=G_stError , 
	Setting:=GVL.stSetting , 
	Recipe:=GVL_Data.stRecipe , 
	Parameter:=_stParameter.stLine3UnloadElevator);
END_ACTION

ACTION A_UnloadLineElevator:
_stParameter.stUnloadLineElevator.bBeltDone:=GVL.I.bFrockBeltDone;
_stParameter.stUnloadLineElevator.bBeltNoneCheck:=GVL.I.bFrockBeltNoneCheck3;
_stParameter.stUnloadLineElevator.bCheck1:=GVL.I.bFrockBeltNoneCheck1;
_stParameter.stUnloadLineElevator.bCheck2:=GVL.I.bFrockBeltNoneCheck2;
_stParameter.stUnloadLineElevator.fbDrive REF= G_arrFbCylinder[E_Cylinder.FrockBelt];
_stParameter.stUnloadLineElevator.fbLineAxis REF= GVL.arrFbLine[E_Line.UnloadElevator];
_stParameter.stUnloadLineElevator.bManualUnload:=FALSE;

_fbUnloadLineElevator(
	Enable:=TRUE,
	System:=G_stSystem , 
	Station:=G_arrStation[E_Station.UnloadLineElevator] , 
	Error:=G_stError , 
	Setting:=GVL.stSetting , 
	Recipe:=GVL_Data.stRecipe , 
	Parameter:=_stParameter.stUnloadLineElevator);
END_ACTION

ACTION A_UnloadLineUc:
_stParameter.stUnloadLineUc.bBeltDone:=GVL.I.bUcBeltDone;
_stParameter.stUnloadLineUc.bBeltNoneCheck:=GVL.I.bUcBeltNoneCheck;
_stParameter.stUnloadLineUc.bCheck1:=GVL.I.bUcCheck2;
_stParameter.stUnloadLineUc.bCheck2:=GVL.I.bUcCheck3;
_stParameter.stUnloadLineUc.fbDrive REF= G_arrFbCylinder[E_Cylinder.UcDrive];
_stParameter.stUnloadLineUc.fbLineAxis REF= GVL.arrFbLine[E_Line.UnloadUC];
_stParameter.stUnloadLineUc.bManualUnload:=FALSE;

_fbUnloadLineUc(
	Enable:=NOT(GVL_Data.stRecipe.eMachineType=E_MachineType.LH311 OR GVL_Data.stRecipe.eMachineType=E_MachineType.RH311),
	System:=G_stSystem , 
	Station:=G_arrStation[E_Station.UnloadLineUc] , 
	Error:=G_stError , 
	Setting:=GVL.stSetting , 
	Recipe:=GVL_Data.stRecipe , 
	Parameter:=_stParameter.stUnloadLineUc);
END_ACTION

ACTION A_UnLoadUc_311:
_stParameter.stUnloadUc_311.bUcCheck1:=GVL.I.bUcCheck1;
_stParameter.stUnloadUc_311.fbAxisY REF= G_arrFbAxis[E_Axis.UC_Y];
_stParameter.stUnloadUc_311.fbClamp REF= G_arrFbCylinder[E_Cylinder.UcClamp];
_stParameter.stUnloadUc_311.fbLift REF= G_arrFbCylinder[E_Cylinder.UcLift];
_stParameter.stUnloadUc_311.fbSwing REF= G_arrFbCylinder[E_Cylinder.UcSwing];

_fbStationUnLoadUc_311(
	Enable:=GVL_Data.stRecipe.eMachineType=E_MachineType.LH311 OR GVL_Data.stRecipe.eMachineType=E_MachineType.RH311,
	System:=G_stSystem , 
	Station:=G_arrStation[E_Station.UnloadUc_311] , 
	Error:=G_stError , 
	Setting:=GVL.stSetting , 
	Recipe:=GVL_Data.stRecipe , 
	Parameter:=_stParameter.stUnloadUc_311);
END_ACTION

ACTION A_UnloadUc_L2:
_stParameter.stLine2UnloadUc.fbClamp REF= G_arrFbCylinder[E_Cylinder.UcClamp1];
_stParameter.stLine2UnloadUc.fbLift REF= G_arrFbCylinder[E_Cylinder.UcLift1];
_stParameter.stLine2UnloadUc.fbRotate REF= G_arrFbCylinder[E_Cylinder.UcRotate1];

_fbUnloadUc_L2(
	Enable:=NOT(GVL_Data.stRecipe.eMachineType=E_MachineType.LH311 OR GVL_Data.stRecipe.eMachineType=E_MachineType.RH311),
	System:=G_stSystem , 
	Station:=G_arrStation[E_Station.Line2UnloadUc] , 
	Error:=G_stError , 
	Setting:=GVL.stSetting , 
	Recipe:=GVL_Data.stRecipe , 
	Parameter:=_stParameter.stLine2UnloadUc);
END_ACTION

ACTION A_UnloadUc_L3:
_stParameter.stLine3UnloadUc.fbClamp REF= G_arrFbCylinder[E_Cylinder.UcClamp2];
_stParameter.stLine3UnloadUc.fbLift REF= G_arrFbCylinder[E_Cylinder.UcLift2];
_stParameter.stLine3UnloadUc.fbRotate REF= G_arrFbCylinder[E_Cylinder.UcRotate2];

	
_fbUnloadUc_L3(
	Enable:=NOT(GVL_Data.stRecipe.eMachineType=E_MachineType.LH311 OR GVL_Data.stRecipe.eMachineType=E_MachineType.RH311),
	System:=G_stSystem , 
	Station:=G_arrStation[E_Station.Line3UnloadUc] , 
	Error:=G_stError , 
	Setting:=GVL.stSetting , 
	Recipe:=GVL_Data.stRecipe , 
	Parameter:=_stParameter.stLine3UnloadUc);
END_ACTION

ACTION A_Virtual:
FOR _i:=0 TO 10 BY 1 DO
	_vArrCylinder[_i].stInput.bHome:=_vArrCylinder[_i].stOutput.bHome;
	_vArrCylinder[_i].stInput.bWork:=_vArrCylinder[_i].stOutput.bWork;
	_vArrFbCylinder[_i](System:=G_stSystem , Cylinder:=_vArrCylinder[_i] , Data:=_vArrCylinderData[_i] , Error:=G_stError );
END_FOR
END_ACTION

METHOD M_LoadPriority : E_TakeMode
VAR_INPUT
	Parameter:		 REFERENCE TO ST_StationParameter;
	Recipe:			 REFERENCE TO ST_Recipe;	
END_VAR
VAR
	_iTemp:					INT;
END_VAR
M_LoadPriority:=E_TakeMode.None;


IF Parameter.stTakeLoad.eState=E_StationState.Done THEN
	IF Parameter.stLine1Load.eState=E_StationState.Load AND Recipe.eLineClose<>E_LineClose.Line2 THEN
		M_LoadPriority:=E_TakeMode.Place1;
	END_IF
	IF Parameter.stLine3Load.eState=E_StationState.Load AND Recipe.eLineClose<>E_LineClose.Line3 THEN
		M_LoadPriority:=E_TakeMode.Place3Load;
	END_IF
END_IF

IF Parameter.stTakeLoad.eState=E_StationState.Load THEN
	IF Parameter.stLine3Load.eState=E_StationState.Done AND Recipe.eLineClose=E_LineClose.Line3 THEN
		M_LoadPriority:=E_TakeMode.Take3Load;
	END_IF
	CASE Recipe.eLoadPriority OF
	E_LoadPriority.None,E_LoadPriority.Line0:
		IF Parameter.stLine1Load.eState=E_StationState.Done AND ((Parameter.stLine3Dismantling.eState=E_StationState.Load AND Parameter.stLine3Load.eState=E_StationState.Load) OR Recipe.eLineClose=E_LineClose.Line2) THEN
			M_LoadPriority:=E_TakeMode.Take1;
		END_IF
		IF Parameter.stLine0Buffer.eState=E_StationState.Done THEN
			M_LoadPriority:=E_TakeMode.Take0;
		END_IF
	E_LoadPriority.Line1:
		IF Parameter.stLine0Buffer.eState=E_StationState.Done THEN
			M_LoadPriority:=E_TakeMode.Take0;
		END_IF
		IF Parameter.stLine1Load.eState=E_StationState.Done AND (Parameter.stLine3Load.eState=E_StationState.Load OR Recipe.eLineClose=E_LineClose.Line2) THEN
			M_LoadPriority:=E_TakeMode.Take1;
		END_IF
	END_CASE
END_IF
END_METHOD

END_PROGRAM

